LIN {X 0,Y 524.018,Z 138.211,A -85,B 0,C 180,E1 -4848.394,E2 -4848.394} C_VEL
LIN {X 0,Y 523.958,Z 138.22,A -85,B 0,C 180,E1 -4851.515,E2 -4851.515} C_VEL
LIN {X 0,Y 524.039,Z 138.205,A -85,B 0,C 180,E1 -4854.613,E2 -4854.613} C_VEL
LIN {X 0,Y 524.109,Z 138.203,A -85,B 0,C 180,E1 -4857.695,E2 -4857.695} C_VEL
LIN {X 0,Y 524.104,Z 138.202,A -85,B 0,C 180,E1 -4860,E2 -4860} C_VEL
LIN {X 0,Y 524.038,Z 138.21,A -85,B 0,C 180,E1 -4863.075,E2 -4863.075} C_VEL
LIN {X 0,Y 524.015,Z 138.212,A -85,B 0,C 180,E1 -4866.16,E2 -4866.16} C_VEL
LIN {X 0,Y 524.035,Z 138.323,A -85,B 0,C 180,E1 -4867.829,E2 -4867.829} C_VEL
LIN {X 0,Y 524.468,Z 143.022,A -85,B 0,C 180,E1 -4868.671,E2 -4868.671} C_VEL
LIN {X 0,Y 524.363,Z 158.584,A -85,B 0,C 180,E1 -4871.402,E2 -4871.402} C_VEL
LIN {X 0,Y 524.251,Z 167.062,A -85,B 0,C 180,E1 -4872.903,E2 -4872.903} C_VEL
LIN {X 0,Y 525.963,Z 177.173,A -85,B 0,C 180,E1 -4873.105,E2 -4873.105} C_VEL
LIN {X 0,Y 525.467,Z 274.512,A -85,B 0,C 180,E1 -4874.499,E2 -4874.499} C_VEL
LIN {X 0,Y 525.258,Z 287.533,A -85,B 0,C 180,E1 -4874.837,E2 -4874.837} C_VEL
LIN {X 0,Y 525.076,Z 300.224,A -85,B 0,C 180,E1 -4875.326,E2 -4875.326} C_VEL
LIN {X 0,Y 524.793,Z 311.875,A -85,B 0,C 180,E1 -4875.935,E2 -4875.935} C_VEL
LIN {X 0,Y 524.491,Z 323.834,A -85,B 0,C 180,E1 -4876.744,E2 -4876.744} C_VEL
LIN {X 0,Y 524.237,Z 334.197,A -85,B 0,C 180,E1 -4877.625,E2 -4877.625} C_VEL
LIN {X 0,Y 524.02,Z 343.233,A -85,B 0,C 180,E1 -4878.574,E2 -4878.574} C_VEL
LIN {X 0,Y 523.804,Z 351.242,A -85,B 0,C 180,E1 -4879.599,E2 -4879.599} C_VEL
LIN {X 0,Y 523.63,Z 359.058,A -85,B 0,C 180,E1 -4880.835,E2 -4880.835} C_VEL
LIN {X 0,Y 523.487,Z 365.471,A -85,B 0,C 180,E1 -4882.126,E2 -4882.126} C_VEL
LIN {X 0,Y 523.444,Z 370.082,A -85,B 0,C 180,E1 -4883.334,E2 -4883.334} C_VEL
LIN {X 0,Y 523.363,Z 373.668,A -85,B 0,C 180,E1 -4884.601,E2 -4884.601} C_VEL
LIN {X 0,Y 523.278,Z 376.084,A -85,B 0,C 180,E1 -4885.86,E2 -4885.86} C_VEL
LIN {X 0,Y 523.276,Z 377.541,A -85,B 0,C 180,E1 -4887.42,E2 -4887.42} C_VEL
LIN {X 0,Y 522.601,Z 377.718,A -85,B 0,C 180,E1 -4888.062,E2 -4888.062} C_VEL
LIN {X 0,Y 519.728,Z 377.402,A -85,B 0,C 180,E1 -4889.105,E2 -4889.105} C_VEL
LIN {X 0,Y 517.322,Z 376.67,A -85,B 0,C 180,E1 -4889.941,E2 -4889.941} C_VEL
LIN {X 0,Y 516.264,Z 375.561,A -85,B 0,C 180,E1 -4890.691,E2 -4890.691} C_VEL
LIN {X 0,Y 516.251,Z 375.333,A -85,B 0,C 180,E1 -4890.799,E2 -4890.799} C_VEL
LIN {X 0,Y 516.301,Z 372.483,A -85,B 0,C 180,E1 -4892.065,E2 -4892.065} C_VEL
LIN {X 0,Y 516.353,Z 368.046,A -85,B 0,C 180,E1 -4893.436,E2 -4893.436} C_VEL
LIN {X 0,Y 516.459,Z 362.961,A -85,B 0,C 180,E1 -4894.621,E2 -4894.621} C_VEL
LIN {X 0,Y 516.626,Z 356.582,A -85,B 0,C 180,E1 -4895.8,E2 -4895.8} C_VEL
LIN {X 0,Y 516.846,Z 348.507,A -85,B 0,C 180,E1 -4896.993,E2 -4896.993} C_VEL
LIN {X 0,Y 517.108,Z 339.432,A -85,B 0,C 180,E1 -4898.077,E2 -4898.077} C_VEL
LIN {X 0,Y 517.351,Z 330.008,A -85,B 0,C 180,E1 -4898.996,E2 -4898.996} C_VEL
LIN {X 0,Y 517.575,Z 320.063,A -85,B 0,C 180,E1 -4899.785,E2 -4899.785} C_VEL
LIN {X 0,Y 517.926,Z 307.968,A -85,B 0,C 180,E1 -4900.545,E2 -4900.545} C_VEL
LIN {X 0,Y 518.248,Z 295.886,A -85,B 0,C 180,E1 -4901.126,E2 -4901.126} C_VEL
LIN {X 0,Y 518.426,Z 282.731,A -85,B 0,C 180,E1 -4901.578,E2 -4901.578} C_VEL
LIN {X 0,Y 518.601,Z 269.587,A -85,B 0,C 180,E1 -4901.862,E2 -4901.862} C_VEL
LIN {X 0,Y 519.056,Z 177.123,A -85,B 0,C 180,E1 -4903.192,E2 -4903.192} C_VEL
LIN {X 0,Y 517.245,Z 167.202,A -85,B 0,C 180,E1 -4903.401,E2 -4903.401} C_VEL
LIN {X 0,Y 517.6,Z 151.206,A -85,B 0,C 180,E1 -4906.433,E2 -4906.433} C_VEL
LIN {X 0,Y 517.694,Z 144.207,A -85,B 0,C 180,E1 -4907.778,E2 -4907.778} C_VEL
LIN {X 0,Y 516.916,Z 139.099,A -85,B 0,C 180,E1 -4908.846,E2 -4908.846} C_VEL
LIN {X 0,Y 516.881,Z 139.099,A -85,B 0,C 180,E1 -4912.058,E2 -4912.058} C_VEL
LIN {X 0,Y 516.877,Z 139.097,A -85,B 0,C 180,E1 -4915.174,E2 -4915.174} C_VEL
LIN {X 0,Y 516.872,Z 139.098,A -85,B 0,C 180,E1 -4917.974,E2 -4917.974} C_VEL
LIN {X 0,Y 516.84,Z 139.105,A -85,B 0,C 180,E1 -4920.69,E2 -4920.69} C_VEL
LIN {X 0,Y 516.839,Z 139.1,A -85,B 0,C 180,E1 -4923.337,E2 -4923.337} C_VEL
LIN {X 0,Y 516.872,Z 139.1,A -85,B 0,C 180,E1 -4925.925,E2 -4925.925} C_VEL
LIN {X 0,Y 516.858,Z 139.104,A -85,B 0,C 180,E1 -4928.46,E2 -4928.46} C_VEL
LIN {X 0,Y 516.868,Z 139.097,A -85,B 0,C 180,E1 -4930.953,E2 -4930.953} C_VEL
LIN {X 0,Y 516.835,Z 139.101,A -85,B 0,C 180,E1 -4933.407,E2 -4933.407} C_VEL
LIN {X 0,Y 516.876,Z 139.101,A -85,B 0,C 180,E1 -4935.832,E2 -4935.832} C_VEL
LIN {X 0,Y 516.931,Z 139.095,A -85,B 0,C 180,E1 -4938.232,E2 -4938.232} C_VEL
LIN {X 0,Y 516.925,Z 139.091,A -85,B 0,C 180,E1 -4941.398,E2 -4941.398} C_VEL
LIN {X 0,Y 516.984,Z 139.083,A -85,B 0,C 180,E1 -4944.539,E2 -4944.539} C_VEL
LIN {X 0,Y 517.077,Z 139.077,A -85,B 0,C 180,E1 -4947.662,E2 -4947.662} C_VEL
LIN {X 0,Y 517.069,Z 139.078,A -85,B 0,C 180,E1 -4949.999,E2 -4949.999} C_VEL
LIN {X 0,Y 517.076,Z 139.072,A -85,B 0,C 180,E1 -4952.336,E2 -4952.336} C_VEL
LIN {X 0,Y 516.982,Z 139.088,A -85,B 0,C 180,E1 -4955.46,E2 -4955.46} C_VEL
LIN {X 0,Y 516.923,Z 139.09,A -85,B 0,C 180,E1 -4958.6,E2 -4958.6} C_VEL
LIN {X 0,Y 516.936,Z 139.094,A -85,B 0,C 180,E1 -4961.795,E2 -4961.795} C_VEL
LIN {X 0,Y 516.938,Z 139.092,A -85,B 0,C 180,E1 -4965.141,E2 -4965.141} C_VEL
LIN {X 0,Y 516.872,Z 139.096,A -85,B 0,C 180,E1 -4968.223,E2 -4968.223} C_VEL
LIN {X 0,Y 516.872,Z 139.097,A -85,B 0,C 180,E1 -4970.702,E2 -4970.702} C_VEL
LIN {X 0,Y 516.841,Z 139.108,A -85,B 0,C 180,E1 -4973.224,E2 -4973.224} C_VEL
LIN {X 0,Y 516.879,Z 139.095,A -85,B 0,C 180,E1 -4976.18,E2 -4976.18} C_VEL
LIN {X 0,Y 516.896,Z 139.101,A -85,B 0,C 180,E1 -4979.305,E2 -4979.305} C_VEL
LIN {X 0,Y 516.891,Z 139.095,A -85,B 0,C 180,E1 -4982.541,E2 -4982.541} C_VEL
LIN {X 0,Y 516.852,Z 139.104,A -85,B 0,C 180,E1 -4985.327,E2 -4985.327} C_VEL
LIN {X 0,Y 516.875,Z 139.096,A -85,B 0,C 180,E1 -4987.941,E2 -4987.941} C_VEL
LIN {X 0,Y 516.847,Z 139.105,A -85,B 0,C 180,E1 -4990.744,E2 -4990.744} C_VEL
LIN {X 0,Y 516.877,Z 139.095,A -85,B 0,C 180,E1 -4993.903,E2 -4993.903} C_VEL
LIN {X 0,Y 516.876,Z 139.096,A -85,B 0,C 180,E1 -4996.106,E2 -4996.106} C_VEL
LIN {X 0,Y 516.843,Z 139.102,A -85,B 0,C 180,E1 -4999.254,E2 -4999.254} C_VEL
LIN {X 0,Y 516.871,Z 139.097,A -85,B 0,C 180,E1 -5002.057,E2 -5002.057} C_VEL
LIN {X 0,Y 516.866,Z 139.099,A -85,B 0,C 180,E1 -5005.173,E2 -5005.173} C_VEL
LIN {X 0,Y 516.861,Z 139.099,A -85,B 0,C 180,E1 -5007.974,E2 -5007.974} C_VEL
LIN {X 0,Y 516.891,Z 139.1,A -85,B 0,C 180,E1 -5010.693,E2 -5010.693} C_VEL
LIN {X 0,Y 516.873,Z 139.097,A -85,B 0,C 180,E1 -5013.818,E2 -5013.818} C_VEL
LIN {X 0,Y 516.835,Z 139.105,A -85,B 0,C 180,E1 -5016.774,E2 -5016.774} C_VEL
LIN {X 0,Y 516.9,Z 139.094,A -85,B 0,C 180,E1 -5019.741,E2 -5019.741} C_VEL
LIN {X 0,Y 516.861,Z 139.102,A -85,B 0,C 180,E1 -5022.593,E2 -5022.593} C_VEL
LIN {X 0,Y 516.923,Z 139.09,A -85,B 0,C 180,E1 -5025.029,E2 -5025.029} C_VEL
LIN {X 0,Y 516.918,Z 139.099,A -85,B 0,C 180,E1 -5028.232,E2 -5028.232} C_VEL
LIN {X 0,Y 516.912,Z 139.092,A -85,B 0,C 180,E1 -5031.398,E2 -5031.398} C_VEL
LIN {X 0,Y 516.976,Z 139.086,A -85,B 0,C 180,E1 -5034.539,E2 -5034.539} C_VEL
LIN {X 0,Y 517.066,Z 139.076,A -85,B 0,C 180,E1 -5037.663,E2 -5037.663} C_VEL
LIN {X 0,Y 517.057,Z 139.081,A -85,B 0,C 180,E1 -5040,E2 -5040} C_VEL
LIN {X 0,Y 517.065,Z 139.075,A -85,B 0,C 180,E1 -5042.337,E2 -5042.337} C_VEL
LIN {X 0,Y 516.96,Z 139.088,A -85,B 0,C 180,E1 -5046.244,E2 -5046.244} C_VEL
LIN {X 0,Y 516.898,Z 139.097,A -85,B 0,C 180,E1 -5049.39,E2 -5049.39} C_VEL
LIN {X 0,Y 516.888,Z 139.094,A -85,B 0,C 180,E1 -5052.565,E2 -5052.565} C_VEL
LIN {X 0,Y 516.927,Z 139.092,A -85,B 0,C 180,E1 -5055.142,E2 -5055.142} C_VEL
LIN {X 0,Y 516.861,Z 139.098,A -85,B 0,C 180,E1 -5058.224,E2 -5058.224} C_VEL
LIN {X 0,Y 516.862,Z 139.098,A -85,B 0,C 180,E1 -5060.704,E2 -5060.704} C_VEL
LIN {X 0,Y 516.831,Z 139.107,A -85,B 0,C 180,E1 -5063.225,E2 -5063.225} C_VEL
LIN {X 0,Y 516.87,Z 139.097,A -85,B 0,C 180,E1 -5066.181,E2 -5066.181} C_VEL
LIN {X 0,Y 516.821,Z 139.102,A -85,B 0,C 180,E1 -5068.421,E2 -5068.421} C_VEL
LIN {X 0,Y 516.84,Z 139.106,A -85,B 0,C 180,E1 -5071.113,E2 -5071.113} C_VEL
LIN {X 0,Y 516.873,Z 139.097,A -85,B 0,C 180,E1 -5073.962,E2 -5073.962} C_VEL
LIN {X 0,Y 516.808,Z 139.107,A -85,B 0,C 180,E1 -5076.752,E2 -5076.752} C_VEL
LIN {X 0,Y 516.849,Z 139.1,A -85,B 0,C 180,E1 -5079.724,E2 -5079.724} C_VEL
LIN {X 0,Y 516.835,Z 139.106,A -85,B 0,C 180,E1 -5082.837,E2 -5082.837} C_VEL
LIN {X 0,Y 516.89,Z 139.103,A -85,B 0,C 180,E1 -5085.008,E2 -5085.008} C_VEL
LIN {X 0,Y 516.842,Z 139.102,A -85,B 0,C 180,E1 -5088.408,E2 -5088.408} C_VEL
LIN {X 0,Y 516.863,Z 139.1,A -85,B 0,C 180,E1 -5091.284,E2 -5091.284} C_VEL
LIN {X 0,Y 516.844,Z 139.107,A -85,B 0,C 180,E1 -5094.674,E2 -5094.674} C_VEL
LIN {X 0,Y 516.863,Z 139.098,A -85,B 0,C 180,E1 -5097.463,E2 -5097.463} C_VEL
LIN {X 0,Y 516.834,Z 139.108,A -85,B 0,C 180,E1 -5100.492,E2 -5100.492} C_VEL
LIN {X 0,Y 516.829,Z 139.105,A -85,B 0,C 180,E1 -5103.338,E2 -5103.338} C_VEL
LIN {X 0,Y 516.887,Z 139.245,A -85,B 0,C 180,E1 -5105.689,E2 -5105.689} C_VEL
LIN {X 0,Y 518.362,Z 147.957,A -85,B 0,C 180,E1 -5107.213,E2 -5107.213} C_VEL
LIN {X 0,Y 517.967,Z 164.813,A -85,B 0,C 180,E1 -5109.975,E2 -5109.975} C_VEL
LIN {X 0,Y 517.491,Z 183.732,A -85,B 0,C 180,E1 -5113.024,E2 -5113.024} C_VEL
LIN {X 0,Y 517.26,Z 194.139,A -85,B 0,C 180,E1 -5114.646,E2 -5114.646} C_VEL
LIN {X 0,Y 518.975,Z 205.188,A -85,B 0,C 180,E1 -5114.86,E2 -5114.86} C_VEL
LIN {X 0,Y 518.55,Z 301.82,A -85,B 0,C 180,E1 -5116.256,E2 -5116.256} C_VEL
LIN {X 0,Y 518.282,Z 315.071,A -85,B 0,C 180,E1 -5116.598,E2 -5116.598} C_VEL
LIN {X 0,Y 518.055,Z 327.249,A -85,B 0,C 180,E1 -5117.066,E2 -5117.066} C_VEL
LIN {X 0,Y 517.752,Z 339.225,A -85,B 0,C 180,E1 -5117.685,E2 -5117.685} C_VEL
LIN {X 0,Y 517.483,Z 350.536,A -85,B 0,C 180,E1 -5118.445,E2 -5118.445} C_VEL
LIN {X 0,Y 517.197,Z 361.119,A -85,B 0,C 180,E1 -5119.331,E2 -5119.331} C_VEL
LIN {X 0,Y 516.924,Z 369.768,A -85,B 0,C 180,E1 -5120.216,E2 -5120.216} C_VEL
LIN {X 0,Y 516.702,Z 377.739,A -85,B 0,C 180,E1 -5121.199,E2 -5121.199} C_VEL
LIN {X 0,Y 516.531,Z 385.528,A -85,B 0,C 180,E1 -5122.377,E2 -5122.377} C_VEL
LIN {X 0,Y 516.384,Z 392.681,A -85,B 0,C 180,E1 -5123.75,E2 -5123.75} C_VEL
LIN {X 0,Y 516.312,Z 397.442,A -85,B 0,C 180,E1 -5124.925,E2 -5124.925} C_VEL
LIN {X 0,Y 516.351,Z 401.081,A -85,B 0,C 180,E1 -5126.098,E2 -5126.098} C_VEL
LIN {X 0,Y 516.282,Z 402.956,A -85,B 0,C 180,E1 -5126.879,E2 -5126.879} C_VEL
LIN {X 0,Y 516.261,Z 404.361,A -85,B 0,C 180,E1 -5127.66,E2 -5127.66} C_VEL
LIN {X 0,Y 516.162,Z 405.969,A -85,B 0,C 180,E1 -5129.221,E2 -5129.221} C_VEL
LIN {X 0,Y 516.159,Z 406.183,A -85,B 0,C 180,E1 -5130.001,E2 -5130.001} C_VEL
LIN {X 0,Y 516.192,Z 405.347,A -85,B 0,C 180,E1 -5131.561,E2 -5131.561} C_VEL
LIN {X 0,Y 516.261,Z 404.34,A -85,B 0,C 180,E1 -5132.341,E2 -5132.341} C_VEL
LIN {X 0,Y 516.282,Z 402.925,A -85,B 0,C 180,E1 -5133.122,E2 -5133.122} C_VEL
LIN {X 0,Y 516.31,Z 399.956,A -85,B 0,C 180,E1 -5134.294,E2 -5134.294} C_VEL
LIN {X 0,Y 516.368,Z 395.937,A -85,B 0,C 180,E1 -5135.468,E2 -5135.468} C_VEL
LIN {X 0,Y 516.463,Z 390.039,A -85,B 0,C 180,E1 -5136.783,E2 -5136.783} C_VEL
LIN {X 0,Y 516.568,Z 382.987,A -85,B 0,C 180,E1 -5138.017,E2 -5138.017} C_VEL
LIN {X 0,Y 516.767,Z 374.592,A -85,B 0,C 180,E1 -5139.196,E2 -5139.196} C_VEL
LIN {X 0,Y 516.988,Z 365.949,A -85,B 0,C 180,E1 -5140.18,E2 -5140.18} C_VEL
LIN {X 0,Y 517.315,Z 355.287,A -85,B 0,C 180,E1 -5141.163,E2 -5141.163} C_VEL
LIN {X 0,Y 517.563,Z 344.395,A -85,B 0,C 180,E1 -5141.974,E2 -5141.974} C_VEL
LIN {X 0,Y 517.885,Z 333.012,A -85,B 0,C 180,E1 -5142.641,E2 -5142.641} C_VEL
LIN {X 0,Y 518.145,Z 320.861,A -85,B 0,C 180,E1 -5143.182,E2 -5143.182} C_VEL
LIN {X 0,Y 518.396,Z 307.676,A -85,B 0,C 180,E1 -5143.6,E2 -5143.6} C_VEL
LIN {X 0,Y 518.58,Z 295.001,A -85,B 0,C 180,E1 -5143.845,E2 -5143.845} C_VEL
LIN {X 0,Y 518.944,Z 204.771,A -85,B 0,C 180,E1 -5145.142,E2 -5145.142} C_VEL
LIN {X 0,Y 517.215,Z 193.411,A -85,B 0,C 180,E1 -5145.369,E2 -5145.369} C_VEL
LIN {X 0,Y 517.695,Z 172.85,A -85,B 0,C 180,E1 -5148.605,E2 -5148.605} C_VEL
LIN {X 0,Y 518.022,Z 154.72,A -85,B 0,C 180,E1 -5151.489,E2 -5151.489} C_VEL
LIN {X 0,Y 518.101,Z 146.04,A -85,B 0,C 180,E1 -5152.893,E2 -5152.893} C_VEL
LIN {X 0,Y 516.868,Z 139.103,A -85,B 0,C 180,E1 -5154.075,E2 -5154.075} C_VEL
LIN {X 0,Y 516.831,Z 139.107,A -85,B 0,C 180,E1 -5156.664,E2 -5156.664} C_VEL
LIN {X 0,Y 516.84,Z 139.107,A -85,B 0,C 180,E1 -5159.509,E2 -5159.509} C_VEL
LIN {X 0,Y 516.87,Z 139.1,A -85,B 0,C 180,E1 -5162.538,E2 -5162.538} C_VEL
LIN {X 0,Y 516.853,Z 139.105,A -85,B 0,C 180,E1 -5165.327,E2 -5165.327} C_VEL
LIN {X 0,Y 516.874,Z 139.102,A -85,B 0,C 180,E1 -5168.717,E2 -5168.717} C_VEL
LIN {X 0,Y 516.848,Z 139.1,A -85,B 0,C 180,E1 -5171.782,E2 -5171.782} C_VEL
LIN {X 0,Y 516.899,Z 139.098,A -85,B 0,C 180,E1 -5175.007,E2 -5175.007} C_VEL
LIN {X 0,Y 516.851,Z 139.102,A -85,B 0,C 180,E1 -5178.407,E2 -5178.407} C_VEL
LIN {X 0,Y 516.876,Z 139.096,A -85,B 0,C 180,E1 -5181.284,E2 -5181.284} C_VEL
LIN {X 0,Y 516.859,Z 139.101,A -85,B 0,C 180,E1 -5184.219,E2 -5184.219} C_VEL
LIN {X 0,Y 516.882,Z 139.098,A -85,B 0,C 180,E1 -5187.052,E2 -5187.052} C_VEL
LIN {X 0,Y 516.849,Z 139.099,A -85,B 0,C 180,E1 -5189.794,E2 -5189.794} C_VEL
LIN {X 0,Y 516.871,Z 139.104,A -85,B 0,C 180,E1 -5192.464,E2 -5192.464} C_VEL
LIN {X 0,Y 516.848,Z 139.1,A -85,B 0,C 180,E1 -5195.069,E2 -5195.069} C_VEL
LIN {X 0,Y 516.873,Z 139.097,A -85,B 0,C 180,E1 -5197.622,E2 -5197.622} C_VEL
LIN {X 0,Y 516.921,Z 139.097,A -85,B 0,C 180,E1 -5200.129,E2 -5200.129} C_VEL
LIN {X 0,Y 516.869,Z 139.1,A -85,B 0,C 180,E1 -5202.594,E2 -5202.594} C_VEL
LIN {X 0,Y 516.944,Z 139.089,A -85,B 0,C 180,E1 -5205.03,E2 -5205.03} C_VEL
LIN {X 0,Y 516.971,Z 139.091,A -85,B 0,C 180,E1 -5208.234,E2 -5208.234} C_VEL
LIN {X 0,Y 516.934,Z 139.093,A -85,B 0,C 180,E1 -5211.399,E2 -5211.399} C_VEL
LIN {X 0,Y 516.99,Z 139.084,A -85,B 0,C 180,E1 -5214.54,E2 -5214.54} C_VEL
LIN {X 0,Y 517.078,Z 139.079,A -85,B 0,C 180,E1 -5217.663,E2 -5217.663} C_VEL
LIN {X 0,Y 517.072,Z 139.078,A -85,B 0,C 180,E1 -5220,E2 -5220} C_VEL
LIN {X 0,Y 517.083,Z 139.074,A -85,B 0,C 180,E1 -5222.337,E2 -5222.337} C_VEL
LIN {X 0,Y 517.015,Z 139.087,A -85,B 0,C 180,E1 -5225.46,E2 -5225.46} C_VEL
LIN {X 0,Y 517.014,Z 139.25,A -85,B 0,C 180,E1 -5227.715,E2 -5227.715} C_VEL
LIN {X 0,Y 517.492,Z 144.098,A -85,B 0,C 180,E1 -5228.592,E2 -5228.592} C_VEL
LIN {X 0,Y 517.391,Z 158.648,A -85,B 0,C 180,E1 -5231.161,E2 -5231.161} C_VEL
LIN {X 0,Y 517.259,Z 167.216,A -85,B 0,C 180,E1 -5232.688,E2 -5232.688} C_VEL
LIN {X 0,Y 519.12,Z 178.22,A -85,B 0,C 180,E1 -5232.919,E2 -5232.919} C_VEL
LIN {X 0,Y 518.548,Z 274.512,A -85,B 0,C 180,E1 -5234.321,E2 -5234.321} C_VEL
LIN {X 0,Y 518.372,Z 287.213,A -85,B 0,C 180,E1 -5234.652,E2 -5234.652} C_VEL
LIN {X 0,Y 518.159,Z 298.618,A -85,B 0,C 180,E1 -5235.084,E2 -5235.084} C_VEL
LIN {X 0,Y 517.918,Z 309.93,A -85,B 0,C 180,E1 -5235.655,E2 -5235.655} C_VEL
LIN {X 0,Y 517.638,Z 320.905,A -85,B 0,C 180,E1 -5236.363,E2 -5236.363} C_VEL
LIN {X 0,Y 517.317,Z 331.088,A -85,B 0,C 180,E1 -5237.187,E2 -5237.187} C_VEL
LIN {X 0,Y 517.068,Z 341.353,A -85,B 0,C 180,E1 -5238.217,E2 -5238.217} C_VEL
LIN {X 0,Y 516.837,Z 349.758,A -85,B 0,C 180,E1 -5239.254,E2 -5239.254} C_VEL
LIN {X 0,Y 516.625,Z 357.334,A -85,B 0,C 180,E1 -5240.406,E2 -5240.406} C_VEL
LIN {X 0,Y 516.465,Z 363.425,A -85,B 0,C 180,E1 -5241.556,E2 -5241.556} C_VEL
LIN {X 0,Y 516.363,Z 368.714,A -85,B 0,C 180,E1 -5242.824,E2 -5242.824} C_VEL
LIN {X 0,Y 516.281,Z 373.025,A -85,B 0,C 180,E1 -5244.208,E2 -5244.208} C_VEL
LIN {X 0,Y 516.236,Z 374.785,A -85,B 0,C 180,E1 -5244.963,E2 -5244.963} C_VEL
LIN {X 0,Y 516.172,Z 376.548,A -85,B 0,C 180,E1 -5246.02,E2 -5246.02} C_VEL
LIN {X 0,Y 516.179,Z 377.719,A -85,B 0,C 180,E1 -5247.422,E2 -5247.422} C_VEL
LIN {X 0,Y 516.187,Z 377.813,A -85,B 0,C 180,E1 -5248.46,E2 -5248.46} C_VEL
LIN {X 0,Y 516.247,Z 377.281,A -85,B 0,C 180,E1 -5249.392,E2 -5249.392} C_VEL
LIN {X 0,Y 516.251,Z 375.333,A -85,B 0,C 180,E1 -5250.799,E2 -5250.799} C_VEL
LIN {X 0,Y 515.62,Z 374.115,A -85,B 0,C 180,E1 -5251.437,E2 -5251.437} C_VEL
LIN {X 0,Y 512.778,Z 371.571,A -85,B 0,C 180,E1 -5252.457,E2 -5252.457} C_VEL
LIN {X 0,Y 510.391,Z 369.044,A -85,B 0,C 180,E1 -5253.261,E2 -5253.261} C_VEL
LIN {X 0,Y 509.413,Z 366.807,A -85,B 0,C 180,E1 -5253.869,E2 -5253.869} C_VEL
LIN {X 0,Y 509.362,Z 365.974,A -85,B 0,C 180,E1 -5254.072,E2 -5254.072} C_VEL
LIN {X 0,Y 509.528,Z 359.589,A -85,B 0,C 180,E1 -5255.403,E2 -5255.403} C_VEL
LIN {X 0,Y 509.71,Z 352.041,A -85,B 0,C 180,E1 -5256.638,E2 -5256.638} C_VEL
LIN {X 0,Y 509.977,Z 343.015,A -85,B 0,C 180,E1 -5257.826,E2 -5257.826} C_VEL
LIN {X 0,Y 510.243,Z 333.745,A -85,B 0,C 180,E1 -5258.808,E2 -5258.808} C_VEL
LIN {X 0,Y 510.548,Z 323.768,A -85,B 0,C 180,E1 -5259.67,E2 -5259.67} C_VEL
LIN {X 0,Y 510.839,Z 313.416,A -85,B 0,C 180,E1 -5260.395,E2 -5260.395} C_VEL
LIN {X 0,Y 511.184,Z 301.901,A -85,B 0,C 180,E1 -5261.033,E2 -5261.033} C_VEL
LIN {X 0,Y 511.397,Z 289.381,A -85,B 0,C 180,E1 -5261.553,E2 -5261.553} C_VEL
LIN {X 0,Y 511.625,Z 276.213,A -85,B 0,C 180,E1 -5261.921,E2 -5261.921} C_VEL
LIN {X 0,Y 511.782,Z 249.363,A -85,B 0,C 180,E1 -5262.341,E2 -5262.341} C_VEL
LIN {X 0,Y 512.117,Z 177.423,A -85,B 0,C 180,E1 -5263.396,E2 -5263.396} C_VEL
LIN {X 0,Y 510.268,Z 167.314,A -85,B 0,C 180,E1 -5263.623,E2 -5263.623} C_VEL
LIN {X 0,Y 510.689,Z 150.589,A -85,B 0,C 180,E1 -5266.835,E2 -5266.835} C_VEL
LIN {X 0,Y 510.672,Z 144.608,A -85,B 0,C 180,E1 -5268.002,E2 -5268.002} C_VEL
LIN {X 0,Y 509.874,Z 139.976,A -85,B 0,C 180,E1 -5268.976,E2 -5268.976} C_VEL
LIN {X 0,Y 509.827,Z 139.976,A -85,B 0,C 180,E1 -5271.791,E2 -5271.791} C_VEL
LIN {X 0,Y 509.824,Z 139.982,A -85,B 0,C 180,E1 -5274.621,E2 -5274.621} C_VEL
LIN {X 0,Y 509.863,Z 139.969,A -85,B 0,C 180,E1 -5277.48,E2 -5277.48} C_VEL
LIN {X 0,Y 509.796,Z 139.984,A -85,B 0,C 180,E1 -5280.287,E2 -5280.287} C_VEL
LIN {X 0,Y 509.824,Z 139.976,A -85,B 0,C 180,E1 -5282.94,E2 -5282.94} C_VEL
LIN {X 0,Y 509.827,Z 139.974,A -85,B 0,C 180,E1 -5285.571,E2 -5285.571} C_VEL
LIN {X 0,Y 509.808,Z 139.983,A -85,B 0,C 180,E1 -5288.147,E2 -5288.147} C_VEL
LIN {X 0,Y 509.83,Z 139.976,A -85,B 0,C 180,E1 -5290.68,E2 -5290.68} C_VEL
LIN {X 0,Y 509.79,Z 139.978,A -85,B 0,C 180,E1 -5293.171,E2 -5293.171} C_VEL
LIN {X 0,Y 509.849,Z 139.973,A -85,B 0,C 180,E1 -5295.633,E2 -5295.633} C_VEL
LIN {X 0,Y 509.895,Z 139.973,A -85,B 0,C 180,E1 -5298.13,E2 -5298.13} C_VEL
LIN {X 0,Y 509.878,Z 139.968,A -85,B 0,C 180,E1 -5301.278,E2 -5301.278} C_VEL
LIN {X 0,Y 509.92,Z 139.967,A -85,B 0,C 180,E1 -5303.669,E2 -5303.669} C_VEL
LIN {X 0,Y 509.888,Z 139.966,A -85,B 0,C 180,E1 -5306.839,E2 -5306.839} C_VEL
LIN {X 0,Y 509.926,Z 139.963,A -85,B 0,C 180,E1 -5308.42,E2 -5308.42} C_VEL
LIN {X 0,Y 510.038,Z 139.953,A -85,B 0,C 180,E1 -5309.999,E2 -5309.999} C_VEL
LIN {X 0,Y 510.044,Z 139.948,A -85,B 0,C 180,E1 -5312.368,E2 -5312.368} C_VEL
LIN {X 0,Y 509.935,Z 139.967,A -85,B 0,C 180,E1 -5315.536,E2 -5315.536} C_VEL
LIN {X 0,Y 509.878,Z 139.972,A -85,B 0,C 180,E1 -5317.922,E2 -5317.922} C_VEL
LIN {X 0,Y 509.864,Z 139.972,A -85,B 0,C 180,E1 -5321.126,E2 -5321.126} C_VEL
LIN {X 0,Y 509.842,Z 139.972,A -85,B 0,C 180,E1 -5324.366,E2 -5324.366} C_VEL
LIN {X 0,Y 509.798,Z 139.979,A -85,B 0,C 180,E1 -5326.827,E2 -5326.827} C_VEL
LIN {X 0,Y 509.827,Z 139.981,A -85,B 0,C 180,E1 -5329.319,E2 -5329.319} C_VEL
LIN {X 0,Y 509.825,Z 139.974,A -85,B 0,C 180,E1 -5332.54,E2 -5332.54} C_VEL
LIN {X 0,Y 509.8,Z 139.986,A -85,B 0,C 180,E1 -5335.299,E2 -5335.299} C_VEL
LIN {X 0,Y 509.81,Z 139.976,A -85,B 0,C 180,E1 -5338.081,E2 -5338.081} C_VEL
LIN {X 0,Y 509.803,Z 139.979,A -85,B 0,C 180,E1 -5340.668,E2 -5340.668} C_VEL
LIN {X 0,Y 509.837,Z 139.976,A -85,B 0,C 180,E1 -5343.462,E2 -5343.462} C_VEL
LIN {X 0,Y 509.801,Z 139.978,A -85,B 0,C 180,E1 -5346.354,E2 -5346.354} C_VEL
LIN {X 0,Y 509.829,Z 139.977,A -85,B 0,C 180,E1 -5349.353,E2 -5349.353} C_VEL
LIN {X 0,Y 509.786,Z 139.982,A -85,B 0,C 180,E1 -5352.494,E2 -5352.494} C_VEL
LIN {X 0,Y 509.836,Z 139.975,A -85,B 0,C 180,E1 -5355.329,E2 -5355.329} C_VEL
LIN {X 0,Y 509.798,Z 139.983,A -85,B 0,C 180,E1 -5358.568,E2 -5358.568} C_VEL
LIN {X 0,Y 509.816,Z 139.975,A -85,B 0,C 180,E1 -5361.658,E2 -5361.658} C_VEL
LIN {X 0,Y 509.813,Z 139.984,A -85,B 0,C 180,E1 -5364.62,E2 -5364.62} C_VEL
LIN {X 0,Y 509.852,Z 139.971,A -85,B 0,C 180,E1 -5367.48,E2 -5367.48} C_VEL
LIN {X 0,Y 509.821,Z 139.979,A -85,B 0,C 180,E1 -5370.279,E2 -5370.279} C_VEL
LIN {X 0,Y 509.812,Z 139.978,A -85,B 0,C 180,E1 -5372.94,E2 -5372.94} C_VEL
LIN {X 0,Y 509.827,Z 139.974,A -85,B 0,C 180,E1 -5375.571,E2 -5375.571} C_VEL
LIN {X 0,Y 509.803,Z 139.982,A -85,B 0,C 180,E1 -5378.147,E2 -5378.147} C_VEL
LIN {X 0,Y 509.837,Z 139.977,A -85,B 0,C 180,E1 -5380.68,E2 -5380.68} C_VEL
LIN {X 0,Y 509.782,Z 139.979,A -85,B 0,C 180,E1 -5383.171,E2 -5383.171} C_VEL
LIN {X 0,Y 509.836,Z 139.974,A -85,B 0,C 180,E1 -5385.633,E2 -5385.633} C_VEL
LIN {X 0,Y 509.882,Z 139.975,A -85,B 0,C 180,E1 -5388.13,E2 -5388.13} C_VEL
LIN {X 0,Y 509.865,Z 139.969,A -85,B 0,C 180,E1 -5391.279,E2 -5391.279} C_VEL
LIN {X 0,Y 509.914,Z 139.966,A -85,B 0,C 180,E1 -5393.669,E2 -5393.669} C_VEL
LIN {X 0,Y 509.877,Z 139.968,A -85,B 0,C 180,E1 -5396.839,E2 -5396.839} C_VEL
LIN {X 0,Y 509.914,Z 139.966,A -85,B 0,C 180,E1 -5398.42,E2 -5398.42} C_VEL
LIN {X 0,Y 510.026,Z 139.957,A -85,B 0,C 180,E1 -5400,E2 -5400} C_VEL
LIN {X 0,Y 510.033,Z 139.95,A -85,B 0,C 180,E1 -5402.369,E2 -5402.369} C_VEL
LIN {X 0,Y 509.927,Z 139.966,A -85,B 0,C 180,E1 -5405.536,E2 -5405.536} C_VEL
LIN {X 0,Y 509.866,Z 139.976,A -85,B 0,C 180,E1 -5407.923,E2 -5407.923} C_VEL
LIN {X 0,Y 509.853,Z 139.972,A -85,B 0,C 180,E1 -5411.127,E2 -5411.127} C_VEL
LIN {X 0,Y 509.815,Z 139.983,A -85,B 0,C 180,E1 -5413.553,E2 -5413.553} C_VEL
LIN {X 0,Y 509.795,Z 139.981,A -85,B 0,C 180,E1 -5416.005,E2 -5416.005} C_VEL
LIN {X 0,Y 509.818,Z 139.975,A -85,B 0,C 180,E1 -5418.485,E2 -5418.485} C_VEL
LIN {X 0,Y 509.809,Z 139.978,A -85,B 0,C 180,E1 -5421.003,E2 -5421.003} C_VEL
LIN {X 0,Y 509.794,Z 139.985,A -85,B 0,C 180,E1 -5423.565,E2 -5423.565} C_VEL
LIN {X 0,Y 509.806,Z 139.976,A -85,B 0,C 180,E1 -5426.356,E2 -5426.356} C_VEL
LIN {X 0,Y 509.785,Z 139.981,A -85,B 0,C 180,E1 -5428.85,E2 -5428.85} C_VEL
LIN {X 0,Y 509.789,Z 139.983,A -85,B 0,C 180,E1 -5431.592,E2 -5431.592} C_VEL
LIN {X 0,Y 509.825,Z 139.974,A -85,B 0,C 180,E1 -5434.415,E2 -5434.415} C_VEL
LIN {X 0,Y 509.775,Z 139.986,A -85,B 0,C 180,E1 -5437.344,E2 -5437.344} C_VEL
LIN {X 0,Y 509.805,Z 139.977,A -85,B 0,C 180,E1 -5440.385,E2 -5440.385} C_VEL
LIN {X 0,Y 509.786,Z 139.981,A -85,B 0,C 180,E1 -5443.575,E2 -5443.575} C_VEL
LIN {X 0,Y 509.786,Z 139.981,A -85,B 0,C 180,E1 -5446.426,E2 -5446.426} C_VEL
LIN {X 0,Y 509.806,Z 139.977,A -85,B 0,C 180,E1 -5449.616,E2 -5449.616} C_VEL
LIN {X 0,Y 509.774,Z 139.986,A -85,B 0,C 180,E1 -5452.657,E2 -5452.657} C_VEL
LIN {X 0,Y 509.834,Z 139.973,A -85,B 0,C 180,E1 -5455.801,E2 -5455.801} C_VEL
LIN {X 0,Y 509.811,Z 139.985,A -85,B 0,C 180,E1 -5458.727,E2 -5458.727} C_VEL
LIN {X 0,Y 509.819,Z 139.977,A -85,B 0,C 180,E1 -5462.051,E2 -5462.051} C_VEL
LIN {X 0,Y 509.792,Z 139.987,A -85,B 0,C 180,E1 -5464.7,E2 -5464.7} C_VEL
LIN {X 0,Y 509.844,Z 140.159,A -85,B 0,C 180,E1 -5465.517,E2 -5465.517} C_VEL
LIN {X 0,Y 511.398,Z 148.702,A -85,B 0,C 180,E1 -5467.038,E2 -5467.038} C_VEL
LIN {X 0,Y 511.037,Z 164.827,A -85,B 0,C 180,E1 -5469.722,E2 -5469.722} C_VEL
LIN {X 0,Y 510.53,Z 181.024,A -85,B 0,C 180,E1 -5472.372,E2 -5472.372} C_VEL
LIN {X 0,Y 510.229,Z 193.684,A -85,B 0,C 180,E1 -5474.423,E2 -5474.423} C_VEL
LIN {X 0,Y 512.14,Z 206.103,A -85,B 0,C 180,E1 -5474.669,E2 -5474.669} C_VEL
LIN {X 0,Y 511.608,Z 302.384,A -85,B 0,C 180,E1 -5476.091,E2 -5476.091} C_VEL
LIN {X 0,Y 511.336,Z 316.131,A -85,B 0,C 180,E1 -5476.463,E2 -5476.463} C_VEL
LIN {X 0,Y 511.1,Z 327.987,A -85,B 0,C 180,E1 -5476.937,E2 -5476.937} C_VEL
LIN {X 0,Y 510.717,Z 340.754,A -85,B 0,C 180,E1 -5477.631,E2 -5477.631} C_VEL
LIN {X 0,Y 510.44,Z 352.83,A -85,B 0,C 180,E1 -5478.485,E2 -5478.485} C_VEL
LIN {X 0,Y 510.156,Z 361.913,A -85,B 0,C 180,E1 -5479.283,E2 -5479.283} C_VEL
LIN {X 0,Y 509.829,Z 371.228,A -85,B 0,C 180,E1 -5480.279,E2 -5480.279} C_VEL
LIN {X 0,Y 509.605,Z 380.27,A -85,B 0,C 180,E1 -5481.475,E2 -5481.475} C_VEL
LIN {X 0,Y 509.426,Z 387.551,A -85,B 0,C 180,E1 -5482.669,E2 -5482.669} C_VEL
LIN {X 0,Y 509.307,Z 392.463,A -85,B 0,C 180,E1 -5483.663,E2 -5483.663} C_VEL
LIN {X 0,Y 509.241,Z 397.233,A -85,B 0,C 180,E1 -5484.854,E2 -5484.854} C_VEL
LIN {X 0,Y 509.244,Z 400.878,A -85,B 0,C 180,E1 -5486.044,E2 -5486.044} C_VEL
LIN {X 0,Y 509.2,Z 402.757,A -85,B 0,C 180,E1 -5486.836,E2 -5486.836} C_VEL
LIN {X 0,Y 509.19,Z 404.166,A -85,B 0,C 180,E1 -5487.628,E2 -5487.628} C_VEL
LIN {X 0,Y 509.076,Z 405.775,A -85,B 0,C 180,E1 -5489.21,E2 -5489.21} C_VEL
LIN {X 0,Y 509.07,Z 405.989,A -85,B 0,C 180,E1 -5490.001,E2 -5490.001} C_VEL
LIN {X 0,Y 509.076,Z 405.766,A -85,B 0,C 180,E1 -5490.792,E2 -5490.792} C_VEL
LIN {X 0,Y 509.19,Z 404.138,A -85,B 0,C 180,E1 -5492.374,E2 -5492.374} C_VEL
LIN {X 0,Y 509.2,Z 402.719,A -85,B 0,C 180,E1 -5493.165,E2 -5493.165} C_VEL
LIN {X 0,Y 509.202,Z 399.741,A -85,B 0,C 180,E1 -5494.354,E2 -5494.354} C_VEL
LIN {X 0,Y 509.284,Z 395.712,A -85,B 0,C 180,E1 -5495.544,E2 -5495.544} C_VEL
LIN {X 0,Y 509.403,Z 389.61,A -85,B 0,C 180,E1 -5496.914,E2 -5496.914} C_VEL
LIN {X 0,Y 509.495,Z 382.727,A -85,B 0,C 180,E1 -5498.129,E2 -5498.129} C_VEL
LIN {X 0,Y 509.725,Z 374.313,A -85,B 0,C 180,E1 -5499.324,E2 -5499.324} C_VEL
LIN {X 0,Y 509.959,Z 365.643,A -85,B 0,C 180,E1 -5500.321,E2 -5500.321} C_VEL
LIN {X 0,Y 510.333,Z 354.953,A -85,B 0,C 180,E1 -5501.318,E2 -5501.318} C_VEL
LIN {X 0,Y 510.602,Z 344.045,A -85,B 0,C 180,E1 -5502.138,E2 -5502.138} C_VEL
LIN {X 0,Y 510.966,Z 331.589,A -85,B 0,C 180,E1 -5502.865,E2 -5502.865} C_VEL
LIN {X 0,Y 511.232,Z 319.076,A -85,B 0,C 180,E1 -5503.415,E2 -5503.415} C_VEL
LIN {X 0,Y 511.505,Z 306.101,A -85,B 0,C 180,E1 -5503.812,E2 -5503.812} C_VEL
LIN {X 0,Y 511.716,Z 290.655,A -85,B 0,C 180,E1 -5504.085,E2 -5504.085} C_VEL
LIN {X 0,Y 511.973,Z 204.978,A -85,B 0,C 180,E1 -5505.346,E2 -5505.346} C_VEL
LIN {X 0,Y 510.214,Z 193.187,A -85,B 0,C 180,E1 -5505.587,E2 -5505.587} C_VEL
LIN {X 0,Y 510.699,Z 173.895,A -85,B 0,C 180,E1 -5508.661,E2 -5508.661} C_VEL
LIN {X 0,Y 511.069,Z 155.803,A -85,B 0,C 180,E1 -5511.584,E2 -5511.584} C_VEL
LIN {X 0,Y 511.183,Z 147.73,A -85,B 0,C 180,E1 -5512.905,E2 -5512.905} C_VEL
LIN {X 0,Y 509.812,Z 139.982,A -85,B 0,C 180,E1 -5514.267,E2 -5514.267} C_VEL
LIN {X 0,Y 509.816,Z 139.985,A -85,B 0,C 180,E1 -5517.06,E2 -5517.06} C_VEL
LIN {X 0,Y 509.786,Z 139.983,A -85,B 0,C 180,E1 -5519.756,E2 -5519.756} C_VEL
LIN {X 0,Y 509.829,Z 139.979,A -85,B 0,C 180,E1 -5522.766,E2 -5522.766} C_VEL
LIN {X 0,Y 509.798,Z 139.981,A -85,B 0,C 180,E1 -5525.574,E2 -5525.574} C_VEL
LIN {X 0,Y 509.817,Z 139.977,A -85,B 0,C 180,E1 -5528.342,E2 -5528.342} C_VEL
LIN {X 0,Y 509.806,Z 139.979,A -85,B 0,C 180,E1 -5531.431,E2 -5531.431} C_VEL
LIN {X 0,Y 509.842,Z 139.978,A -85,B 0,C 180,E1 -5534.67,E2 -5534.67} C_VEL
LIN {X 0,Y 509.791,Z 139.978,A -85,B 0,C 180,E1 -5537.506,E2 -5537.506} C_VEL
LIN {X 0,Y 509.833,Z 139.98,A -85,B 0,C 180,E1 -5540.646,E2 -5540.646} C_VEL
LIN {X 0,Y 509.805,Z 139.976,A -85,B 0,C 180,E1 -5543.645,E2 -5543.645} C_VEL
LIN {X 0,Y 509.841,Z 139.979,A -85,B 0,C 180,E1 -5546.538,E2 -5546.538} C_VEL
LIN {X 0,Y 509.823,Z 139.974,A -85,B 0,C 180,E1 -5549.333,E2 -5549.333} C_VEL
LIN {X 0,Y 509.827,Z 139.977,A -85,B 0,C 180,E1 -5552.051,E2 -5552.051} C_VEL
LIN {X 0,Y 509.804,Z 139.98,A -85,B 0,C 180,E1 -5554.7,E2 -5554.7} C_VEL
LIN {X 0,Y 509.828,Z 139.974,A -85,B 0,C 180,E1 -5557.459,E2 -5557.459} C_VEL
LIN {X 0,Y 509.909,Z 139.967,A -85,B 0,C 180,E1 -5559.844,E2 -5559.844} C_VEL
LIN {X 0,Y 509.85,Z 139.978,A -85,B 0,C 180,E1 -5562.347,E2 -5562.347} C_VEL
LIN {X 0,Y 509.893,Z 139.968,A -85,B 0,C 180,E1 -5564.818,E2 -5564.818} C_VEL
LIN {X 0,Y 509.905,Z 139.972,A -85,B 0,C 180,E1 -5568.124,E2 -5568.124} C_VEL
LIN {X 0,Y 509.888,Z 139.97,A -85,B 0,C 180,E1 -5571.279,E2 -5571.279} C_VEL
LIN {X 0,Y 509.944,Z 139.962,A -85,B 0,C 180,E1 -5574.464,E2 -5574.464} C_VEL
LIN {X 0,Y 510.047,Z 139.955,A -85,B 0,C 180,E1 -5577.631,E2 -5577.631} C_VEL
LIN {X 0,Y 510.041,Z 139.954,A -85,B 0,C 180,E1 -5580,E2 -5580} C_VEL
LIN {X 0,Y 510.052,Z 139.95,A -85,B 0,C 180,E1 -5582.369,E2 -5582.369} C_VEL
LIN {X 0,Y 509.966,Z 139.965,A -85,B 0,C 180,E1 -5585.536,E2 -5585.536} C_VEL
LIN {X 0,Y 509.954,Z 140.148,A -85,B 0,C 180,E1 -5587.573,E2 -5587.573} C_VEL
LIN {X 0,Y 510.531,Z 145.232,A -85,B 0,C 180,E1 -5588.51,E2 -5588.51} C_VEL
LIN {X 0,Y 510.395,Z 159.842,A -85,B 0,C 180,E1 -5591.115,E2 -5591.115} C_VEL
LIN {X 0,Y 510.345,Z 167.687,A -85,B 0,C 180,E1 -5592.486,E2 -5592.486} C_VEL
LIN {X 0,Y 512.286,Z 179.682,A -85,B 0,C 180,E1 -5592.73,E2 -5592.73} C_VEL
LIN {X 0,Y 511.657,Z 274.521,A -85,B 0,C 180,E1 -5594.137,E2 -5594.137} C_VEL
LIN {X 0,Y 511.45,Z 287.306,A -85,B 0,C 180,E1 -5594.473,E2 -5594.473} C_VEL
LIN {X 0,Y 511.208,Z 300.471,A -85,B 0,C 180,E1 -5594.989,E2 -5594.989} C_VEL
LIN {X 0,Y 510.892,Z 312.657,A -85,B 0,C 180,E1 -5595.645,E2 -5595.645} C_VEL
LIN {X 0,Y 510.531,Z 324.791,A -85,B 0,C 180,E1 -5596.495,E2 -5596.495} C_VEL
LIN {X 0,Y 510.203,Z 335.385,A -85,B 0,C 180,E1 -5597.434,E2 -5597.434} C_VEL
LIN {X 0,Y 509.939,Z 344.871,A -85,B 0,C 180,E1 -5598.481,E2 -5598.481} C_VEL
LIN {X 0,Y 509.701,Z 352.684,A -85,B 0,C 180,E1 -5599.535,E2 -5599.535} C_VEL
LIN {X 0,Y 509.491,Z 360.378,A -85,B 0,C 180,E1 -5600.818,E2 -5600.818} C_VEL
LIN {X 0,Y 509.331,Z 366.534,A -85,B 0,C 180,E1 -5602.139,E2 -5602.139} C_VEL
LIN {X 0,Y 509.222,Z 371.673,A -85,B 0,C 180,E1 -5603.594,E2 -5603.594} C_VEL
LIN {X 0,Y 509.174,Z 373.956,A -85,B 0,C 180,E1 -5604.462,E2 -5604.462} C_VEL
LIN {X 0,Y 509.11,Z 375.74,A -85,B 0,C 180,E1 -5605.337,E2 -5605.337} C_VEL
LIN {X 0,Y 509.099,Z 377.028,A -85,B 0,C 180,E1 -5606.216,E2 -5606.216} C_VEL
LIN {X 0,Y 509.078,Z 377.787,A -85,B 0,C 180,E1 -5607.102,E2 -5607.102} C_VEL
LIN {X 0,Y 509.089,Z 378.085,A -85,B 0,C 180,E1 -5607.994,E2 -5607.994} C_VEL
LIN {X 0,Y 509.139,Z 377.298,A -85,B 0,C 180,E1 -5609.583,E2 -5609.583} C_VEL
LIN {X 0,Y 509.199,Z 374.951,A -85,B 0,C 180,E1 -5611.159,E2 -5611.159} C_VEL
LIN {X 0,Y 509.228,Z 371.106,A -85,B 0,C 180,E1 -5612.66,E2 -5612.66} C_VEL
LIN {X 0,Y 509.362,Z 365.974,A -85,B 0,C 180,E1 -5614.072,E2 -5614.072} C_VEL
LIN {X 0,Y 508.791,Z 363.434,A -85,B 0,C 180,E1 -5614.669,E2 -5614.669} C_VEL
LIN {X 0,Y 506.069,Z 358.889,A -85,B 0,C 180,E1 -5615.616,E2 -5615.616} C_VEL
LIN {X 0,Y 503.341,Z 353.679,A -85,B 0,C 180,E1 -5616.526,E2 -5616.526} C_VEL
LIN {X 0,Y 502.768,Z 350.094,A -85,B 0,C 180,E1 -5617.059,E2 -5617.059} C_VEL
LIN {X 0,Y 503.02,Z 341.444,A -85,B 0,C 180,E1 -5618.155,E2 -5618.155} C_VEL
LIN {X 0,Y 503.335,Z 331.431,A -85,B 0,C 180,E1 -5619.185,E2 -5619.185} C_VEL
LIN {X 0,Y 503.639,Z 320.826,A -85,B 0,C 180,E1 -5620.065,E2 -5620.065} C_VEL
LIN {X 0,Y 504.019,Z 309.339,A -85,B 0,C 180,E1 -5620.816,E2 -5620.816} C_VEL
LIN {X 0,Y 504.364,Z 297.39,A -85,B 0,C 180,E1 -5621.42,E2 -5621.42} C_VEL
LIN {X 0,Y 504.575,Z 285.264,A -85,B 0,C 180,E1 -5621.873,E2 -5621.873} C_VEL
LIN {X 0,Y 504.774,Z 272.092,A -85,B 0,C 180,E1 -5622.191,E2 -5622.191} C_VEL
LIN {X 0,Y 505.283,Z 178.343,A -85,B 0,C 180,E1 -5623.591,E2 -5623.591} C_VEL
LIN {X 0,Y 503.28,Z 167.512,A -85,B 0,C 180,E1 -5623.833,E2 -5623.833} C_VEL
LIN {X 0,Y 503.768,Z 150.718,A -85,B 0,C 180,E1 -5627.097,E2 -5627.097} C_VEL
LIN {X 0,Y 503.59,Z 145.114,A -85,B 0,C 180,E1 -5628.21,E2 -5628.21} C_VEL
LIN {X 0,Y 502.836,Z 140.852,A -85,B 0,C 180,E1 -5629.114,E2 -5629.114} C_VEL
LIN {X 0,Y 502.777,Z 140.856,A -85,B 0,C 180,E1 -5632.044,E2 -5632.044} C_VEL
LIN {X 0,Y 502.794,Z 140.852,A -85,B 0,C 180,E1 -5635.033,E2 -5635.033} C_VEL
LIN {X 0,Y 502.784,Z 140.853,A -85,B 0,C 180,E1 -5637.915,E2 -5637.915} C_VEL
LIN {X 0,Y 502.763,Z 140.858,A -85,B 0,C 180,E1 -5640.708,E2 -5640.708} C_VEL
LIN {X 0,Y 502.777,Z 140.852,A -85,B 0,C 180,E1 -5643.46,E2 -5643.46} C_VEL
LIN {X 0,Y 502.758,Z 140.86,A -85,B 0,C 180,E1 -5646.084,E2 -5646.084} C_VEL
LIN {X 0,Y 502.764,Z 140.856,A -85,B 0,C 180,E1 -5648.687,E2 -5648.687} C_VEL
LIN {X 0,Y 502.798,Z 140.854,A -85,B 0,C 180,E1 -5651.897,E2 -5651.897} C_VEL
LIN {X 0,Y 502.83,Z 140.846,A -85,B 0,C 180,E1 -5655.428,E2 -5655.428} C_VEL
LIN {X 0,Y 502.842,Z 140.845,A -85,B 0,C 180,E1 -5658.715,E2 -5658.715} C_VEL
LIN {X 0,Y 502.851,Z 140.852,A -85,B 0,C 180,E1 -5661.965,E2 -5661.965} C_VEL
LIN {X 0,Y 502.896,Z 140.84,A -85,B 0,C 180,E1 -5664.385,E2 -5664.385} C_VEL
LIN {X 0,Y 503.013,Z 140.828,A -85,B 0,C 180,E1 -5667.597,E2 -5667.597} C_VEL
LIN {X 0,Y 503.007,Z 140.829,A -85,B 0,C 180,E1 -5669.999,E2 -5669.999} C_VEL
LIN {X 0,Y 503.012,Z 140.824,A -85,B 0,C 180,E1 -5672.402,E2 -5672.402} C_VEL
LIN {X 0,Y 502.891,Z 140.846,A -85,B 0,C 180,E1 -5675.613,E2 -5675.613} C_VEL
LIN {X 0,Y 502.85,Z 140.846,A -85,B 0,C 180,E1 -5678.033,E2 -5678.033} C_VEL
LIN {X 0,Y 502.84,Z 140.849,A -85,B 0,C 180,E1 -5681.283,E2 -5681.283} C_VEL
LIN {X 0,Y 502.824,Z 140.846,A -85,B 0,C 180,E1 -5684.571,E2 -5684.571} C_VEL
LIN {X 0,Y 502.786,Z 140.853,A -85,B 0,C 180,E1 -5687.909,E2 -5687.909} C_VEL
LIN {X 0,Y 502.804,Z 140.849,A -85,B 0,C 180,E1 -5690.527,E2 -5690.527} C_VEL
LIN {X 0,Y 502.782,Z 140.856,A -85,B 0,C 180,E1 -5693.04,E2 -5693.04} C_VEL
LIN {X 0,Y 502.776,Z 140.855,A -85,B 0,C 180,E1 -5695.678,E2 -5695.678} C_VEL
LIN {X 0,Y 502.769,Z 140.853,A -85,B 0,C 180,E1 -5698.376,E2 -5698.376} C_VEL
LIN {X 0,Y 502.764,Z 140.862,A -85,B 0,C 180,E1 -5701.145,E2 -5701.145} C_VEL
LIN {X 0,Y 502.784,Z 140.851,A -85,B 0,C 180,E1 -5703.994,E2 -5703.994} C_VEL
LIN {X 0,Y 502.761,Z 140.861,A -85,B 0,C 180,E1 -5707.174,E2 -5707.174} C_VEL
LIN {X 0,Y 502.768,Z 140.853,A -85,B 0,C 180,E1 -5710.016,E2 -5710.016} C_VEL
LIN {X 0,Y 502.743,Z 140.86,A -85,B 0,C 180,E1 -5713.233,E2 -5713.233} C_VEL
LIN {X 0,Y 502.775,Z 140.853,A -85,B 0,C 180,E1 -5715.659,E2 -5715.659} C_VEL
LIN {X 0,Y 502.758,Z 140.86,A -85,B 0,C 180,E1 -5719.012,E2 -5719.012} C_VEL
LIN {X 0,Y 502.767,Z 140.854,A -85,B 0,C 180,E1 -5722.043,E2 -5722.043} C_VEL
LIN {X 0,Y 502.783,Z 140.855,A -85,B 0,C 180,E1 -5725.032,E2 -5725.032} C_VEL
LIN {X 0,Y 502.773,Z 140.853,A -85,B 0,C 180,E1 -5727.914,E2 -5727.914} C_VEL
LIN {X 0,Y 502.783,Z 140.858,A -85,B 0,C 180,E1 -5730.709,E2 -5730.709} C_VEL
LIN {X 0,Y 502.767,Z 140.853,A -85,B 0,C 180,E1 -5733.459,E2 -5733.459} C_VEL
LIN {X 0,Y 502.754,Z 140.859,A -85,B 0,C 180,E1 -5736.084,E2 -5736.084} C_VEL
LIN {X 0,Y 502.823,Z 140.846,A -85,B 0,C 180,E1 -5739.463,E2 -5739.463} C_VEL
LIN {X 0,Y 502.777,Z 140.857,A -85,B 0,C 180,E1 -5742.09,E2 -5742.09} C_VEL
LIN {X 0,Y 502.817,Z 140.847,A -85,B 0,C 180,E1 -5745.428,E2 -5745.428} C_VEL
LIN {X 0,Y 502.83,Z 140.847,A -85,B 0,C 180,E1 -5748.715,E2 -5748.715} C_VEL
LIN {X 0,Y 502.838,Z 140.851,A -85,B 0,C 180,E1 -5751.965,E2 -5751.965} C_VEL
LIN {X 0,Y 502.888,Z 140.842,A -85,B 0,C 180,E1 -5754.386,E2 -5754.386} C_VEL
LIN {X 0,Y 503.001,Z 140.827,A -85,B 0,C 180,E1 -5757.597,E2 -5757.597} C_VEL
LIN {X 0,Y 502.995,Z 140.833,A -85,B 0,C 180,E1 -5760,E2 -5760} C_VEL
LIN {X 0,Y 503.001,Z 140.826,A -85,B 0,C 180,E1 -5762.402,E2 -5762.402} C_VEL
LIN {X 0,Y 502.884,Z 140.844,A -85,B 0,C 180,E1 -5765.614,E2 -5765.614} C_VEL
LIN {X 0,Y 502.838,Z 140.849,A -85,B 0,C 180,E1 -5768.034,E2 -5768.034} C_VEL
LIN {X 0,Y 502.828,Z 140.849,A -85,B 0,C 180,E1 -5771.284,E2 -5771.284} C_VEL
LIN {X 0,Y 502.815,Z 140.847,A -85,B 0,C 180,E1 -5774.572,E2 -5774.572} C_VEL
LIN {X 0,Y 502.776,Z 140.856,A -85,B 0,C 180,E1 -5777.91,E2 -5777.91} C_VEL
LIN {X 0,Y 502.794,Z 140.85,A -85,B 0,C 180,E1 -5780.528,E2 -5780.528} C_VEL
LIN {X 0,Y 502.771,Z 140.856,A -85,B 0,C 180,E1 -5783.042,E2 -5783.042} C_VEL
LIN {X 0,Y 502.767,Z 140.858,A -85,B 0,C 180,E1 -5785.68,E2 -5785.68} C_VEL
LIN {X 0,Y 502.751,Z 140.855,A -85,B 0,C 180,E1 -5788.378,E2 -5788.378} C_VEL
LIN {X 0,Y 502.763,Z 140.859,A -85,B 0,C 180,E1 -5791.495,E2 -5791.495} C_VEL
LIN {X 0,Y 502.778,Z 140.852,A -85,B 0,C 180,E1 -5794.441,E2 -5794.441} C_VEL
LIN {X 0,Y 502.729,Z 140.867,A -85,B 0,C 180,E1 -5797.172,E2 -5797.172} C_VEL
LIN {X 0,Y 502.762,Z 140.854,A -85,B 0,C 180,E1 -5800.018,E2 -5800.018} C_VEL
LIN {X 0,Y 502.733,Z 140.863,A -85,B 0,C 180,E1 -5803.236,E2 -5803.236} C_VEL
LIN {X 0,Y 502.761,Z 140.855,A -85,B 0,C 180,E1 -5805.659,E2 -5805.659} C_VEL
LIN {X 0,Y 502.756,Z 140.862,A -85,B 0,C 180,E1 -5809.013,E2 -5809.013} C_VEL
LIN {X 0,Y 502.754,Z 140.855,A -85,B 0,C 180,E1 -5812.044,E2 -5812.044} C_VEL
LIN {X 0,Y 502.777,Z 140.857,A -85,B 0,C 180,E1 -5815.033,E2 -5815.033} C_VEL
LIN {X 0,Y 502.754,Z 140.855,A -85,B 0,C 180,E1 -5817.914,E2 -5817.914} C_VEL
LIN {X 0,Y 502.749,Z 140.863,A -85,B 0,C 180,E1 -5820.708,E2 -5820.708} C_VEL
LIN {X 0,Y 502.769,Z 140.857,A -85,B 0,C 180,E1 -5823.461,E2 -5823.461} C_VEL
LIN {X 0,Y 502.775,Z 140.901,A -85,B 0,C 180,E1 -5825.312,E2 -5825.312} C_VEL
LIN {X 0,Y 504.46,Z 150.485,A -85,B 0,C 180,E1 -5827.041,E2 -5827.041} C_VEL
LIN {X 0,Y 504.066,Z 165.68,A -85,B 0,C 180,E1 -5829.601,E2 -5829.601} C_VEL
LIN {X 0,Y 503.587,Z 180.845,A -85,B 0,C 180,E1 -5832.121,E2 -5832.121} C_VEL
LIN {X 0,Y 503.257,Z 193.529,A -85,B 0,C 180,E1 -5834.205,E2 -5834.205} C_VEL
LIN {X 0,Y 505.275,Z 207.711,A -85,B 0,C 180,E1 -5834.486,E2 -5834.486} C_VEL
LIN {X 0,Y 504.733,Z 301.779,A -85,B 0,C 180,E1 -5835.897,E2 -5835.897} C_VEL
LIN {X 0,Y 504.451,Z 314.899,A -85,B 0,C 180,E1 -5836.249,E2 -5836.249} C_VEL
LIN {X 0,Y 504.149,Z 327.585,A -85,B 0,C 180,E1 -5836.754,E2 -5836.754} C_VEL
LIN {X 0,Y 503.809,Z 339.065,A -85,B 0,C 180,E1 -5837.371,E2 -5837.371} C_VEL
LIN {X 0,Y 503.486,Z 351.227,A -85,B 0,C 180,E1 -5838.221,E2 -5838.221} C_VEL
LIN {X 0,Y 503.164,Z 361.633,A -85,B 0,C 180,E1 -5839.132,E2 -5839.132} C_VEL
LIN {X 0,Y 502.805,Z 370.972,A -85,B 0,C 180,E1 -5840.142,E2 -5840.142} C_VEL
LIN {X 0,Y 502.551,Z 380.029,A -85,B 0,C 180,E1 -5841.354,E2 -5841.354} C_VEL
LIN {X 0,Y 502.342,Z 387.322,A -85,B 0,C 180,E1 -5842.565,E2 -5842.565} C_VEL
LIN {X 0,Y 502.234,Z 392.245,A -85,B 0,C 180,E1 -5843.573,E2 -5843.573} C_VEL
LIN {X 0,Y 502.171,Z 397.025,A -85,B 0,C 180,E1 -5844.781,E2 -5844.781} C_VEL
LIN {X 0,Y 502.137,Z 400.676,A -85,B 0,C 180,E1 -5845.988,E2 -5845.988} C_VEL
LIN {X 0,Y 502.12,Z 402.559,A -85,B 0,C 180,E1 -5846.791,E2 -5846.791} C_VEL
LIN {X 0,Y 502.092,Z 403.97,A -85,B 0,C 180,E1 -5847.594,E2 -5847.594} C_VEL
LIN {X 0,Y 501.992,Z 405.581,A -85,B 0,C 180,E1 -5849.199,E2 -5849.199} C_VEL
LIN {X 0,Y 501.984,Z 405.795,A -85,B 0,C 180,E1 -5850.001,E2 -5850.001} C_VEL
LIN {X 0,Y 501.993,Z 405.571,A -85,B 0,C 180,E1 -5850.803,E2 -5850.803} C_VEL
LIN {X 0,Y 502.092,Z 403.936,A -85,B 0,C 180,E1 -5852.407,E2 -5852.407} C_VEL
LIN {X 0,Y 502.12,Z 402.513,A -85,B 0,C 180,E1 -5853.21,E2 -5853.21} C_VEL
LIN {X 0,Y 502.1,Z 399.526,A -85,B 0,C 180,E1 -5854.416,E2 -5854.416} C_VEL
LIN {X 0,Y 502.199,Z 395.487,A -85,B 0,C 180,E1 -5855.622,E2 -5855.622} C_VEL
LIN {X 0,Y 502.33,Z 389.366,A -85,B 0,C 180,E1 -5857.012,E2 -5857.012} C_VEL
LIN {X 0,Y 502.448,Z 382.469,A -85,B 0,C 180,E1 -5858.244,E2 -5858.244} C_VEL
LIN {X 0,Y 502.69,Z 374.036,A -85,B 0,C 180,E1 -5859.456,E2 -5859.456} C_VEL
LIN {X 0,Y 502.95,Z 365.343,A -85,B 0,C 180,E1 -5860.467,E2 -5860.467} C_VEL
LIN {X 0,Y 503.33,Z 354.631,A -85,B 0,C 180,E1 -5861.478,E2 -5861.478} C_VEL
LIN {X 0,Y 503.606,Z 344.269,A -85,B 0,C 180,E1 -5862.269,E2 -5862.269} C_VEL
LIN {X 0,Y 504.006,Z 332.185,A -85,B 0,C 180,E1 -5862.995,E2 -5862.995} C_VEL
LIN {X 0,Y 504.292,Z 319.919,A -85,B 0,C 180,E1 -5863.551,E2 -5863.551} C_VEL
LIN {X 0,Y 504.588,Z 306.547,A -85,B 0,C 180,E1 -5863.98,E2 -5863.98} C_VEL
LIN {X 0,Y 504.809,Z 291.614,A -85,B 0,C 180,E1 -5864.256,E2 -5864.256} C_VEL
LIN {X 0,Y 505.165,Z 205.913,A -85,B 0,C 180,E1 -5865.543,E2 -5865.543} C_VEL
LIN {X 0,Y 503.203,Z 192.921,A -85,B 0,C 180,E1 -5865.818,E2 -5865.818} C_VEL
LIN {X 0,Y 503.703,Z 173.701,A -85,B 0,C 180,E1 -5868.93,E2 -5868.93} C_VEL
LIN {X 0,Y 504.112,Z 156.886,A -85,B 0,C 180,E1 -5871.682,E2 -5871.682} C_VEL
LIN {X 0,Y 504.176,Z 148.504,A -85,B 0,C 180,E1 -5873.072,E2 -5873.072} C_VEL
LIN {X 0,Y 502.787,Z 140.857,A -85,B 0,C 180,E1 -5874.444,E2 -5874.444} C_VEL
LIN {X 0,Y 502.771,Z 140.863,A -85,B 0,C 180,E1 -5877.471,E2 -5877.471} C_VEL
LIN {X 0,Y 502.745,Z 140.858,A -85,B 0,C 180,E1 -5880.216,E2 -5880.216} C_VEL
LIN {X 0,Y 502.801,Z 140.857,A -85,B 0,C 180,E1 -5883.034,E2 -5883.034} C_VEL
LIN {X 0,Y 502.749,Z 140.857,A -85,B 0,C 180,E1 -5885.954,E2 -5885.954} C_VEL
LIN {X 0,Y 502.784,Z 140.86,A -85,B 0,C 180,E1 -5888.978,E2 -5888.978} C_VEL
LIN {X 0,Y 502.747,Z 140.857,A -85,B 0,C 180,E1 -5892.192,E2 -5892.192} C_VEL
LIN {X 0,Y 502.788,Z 140.851,A -85,B 0,C 180,E1 -5895.47,E2 -5895.47} C_VEL
LIN {X 0,Y 502.764,Z 140.858,A -85,B 0,C 180,E1 -5898.928,E2 -5898.928} C_VEL
LIN {X 0,Y 502.774,Z 140.853,A -85,B 0,C 180,E1 -5902.044,E2 -5902.044} C_VEL
LIN {X 0,Y 502.791,Z 140.854,A -85,B 0,C 180,E1 -5905.034,E2 -5905.034} C_VEL
LIN {X 0,Y 502.781,Z 140.854,A -85,B 0,C 180,E1 -5907.915,E2 -5907.915} C_VEL
LIN {X 0,Y 502.792,Z 140.854,A -85,B 0,C 180,E1 -5910.71,E2 -5910.71} C_VEL
LIN {X 0,Y 502.777,Z 140.853,A -85,B 0,C 180,E1 -5913.46,E2 -5913.46} C_VEL
LIN {X 0,Y 502.77,Z 140.859,A -85,B 0,C 180,E1 -5916.085,E2 -5916.085} C_VEL
LIN {X 0,Y 502.781,Z 140.853,A -85,B 0,C 180,E1 -5918.689,E2 -5918.689} C_VEL
LIN {X 0,Y 502.81,Z 140.849,A -85,B 0,C 180,E1 -5921.248,E2 -5921.248} C_VEL
LIN {X 0,Y 502.84,Z 140.847,A -85,B 0,C 180,E1 -5924.665,E2 -5924.665} C_VEL
LIN {X 0,Y 502.881,Z 140.847,A -85,B 0,C 180,E1 -5928.039,E2 -5928.039} C_VEL
LIN {X 0,Y 502.853,Z 140.846,A -85,B 0,C 180,E1 -5931.156,E2 -5931.156} C_VEL
LIN {X 0,Y 502.873,Z 140.848,A -85,B 0,C 180,E1 -5933.581,E2 -5933.581} C_VEL
LIN {X 0,Y 502.839,Z 140.846,A -85,B 0,C 180,E1 -5936.795,E2 -5936.795} C_VEL
LIN {X 0,Y 502.897,Z 140.84,A -85,B 0,C 180,E1 -5938.399,E2 -5938.399} C_VEL
LIN {X 0,Y 503.01,Z 140.831,A -85,B 0,C 180,E1 -5940,E2 -5940} C_VEL
LIN {X 0,Y 503.021,Z 140.826,A -85,B 0,C 180,E1 -5942.402,E2 -5942.402} C_VEL
LIN {X 0,Y 502.92,Z 140.843,A -85,B 0,C 180,E1 -5945.614,E2 -5945.614} C_VEL
LIN {X 0,Y 502.913,Z 140.926,A -85,B 0,C 180,E1 -5947.402,E2 -5947.402} C_VEL
LIN {X 0,Y 503.582,Z 146.456,A -85,B 0,C 180,E1 -5948.427,E2 -5948.427} C_VEL
LIN {X 0,Y 503.428,Z 161.071,A -85,B 0,C 180,E1 -5951.067,E2 -5951.067} C_VEL
LIN {X 0,Y 503.371,Z 167.897,A -85,B 0,C 180,E1 -5952.26,E2 -5952.26} C_VEL
LIN {X 0,Y 505.456,Z 180.308,A -85,B 0,C 180,E1 -5952.523,E2 -5952.523} C_VEL
LIN {X 0,Y 504.728,Z 275.816,A -85,B 0,C 180,E1 -5953.975,E2 -5953.975} C_VEL
LIN {X 0,Y 504.5,Z 289.001,A -85,B 0,C 180,E1 -5954.342,E2 -5954.342} C_VEL
LIN {X 0,Y 504.269,Z 301.168,A -85,B 0,C 180,E1 -5954.839,E2 -5954.839} C_VEL
LIN {X 0,Y 503.967,Z 312.574,A -85,B 0,C 180,E1 -5955.463,E2 -5955.463} C_VEL
LIN {X 0,Y 503.569,Z 324.62,A -85,B 0,C 180,E1 -5956.313,E2 -5956.313} C_VEL
LIN {X 0,Y 503.225,Z 335.304,A -85,B 0,C 180,E1 -5957.264,E2 -5957.264} C_VEL
LIN {X 0,Y 502.972,Z 343.536,A -85,B 0,C 180,E1 -5958.164,E2 -5958.164} C_VEL
LIN {X 0,Y 502.656,Z 352.7,A -85,B 0,C 180,E1 -5959.395,E2 -5959.395} C_VEL
LIN {X 0,Y 502.44,Z 360.372,A -85,B 0,C 180,E1 -5960.683,E2 -5960.683} C_VEL
LIN {X 0,Y 502.332,Z 365.509,A -85,B 0,C 180,E1 -5961.763,E2 -5961.763} C_VEL
LIN {X 0,Y 502.194,Z 370.431,A -85,B 0,C 180,E1 -5963.07,E2 -5963.07} C_VEL
LIN {X 0,Y 502.096,Z 374.381,A -85,B 0,C 180,E1 -5964.518,E2 -5964.518} C_VEL
LIN {X 0,Y 502.006,Z 376.597,A -85,B 0,C 180,E1 -5965.722,E2 -5965.722} C_VEL
LIN {X 0,Y 502.001,Z 377.644,A -85,B 0,C 180,E1 -5966.616,E2 -5966.616} C_VEL
LIN {X 0,Y 501.988,Z 378.277,A -85,B 0,C 180,E1 -5968.112,E2 -5968.112} C_VEL
LIN {X 0,Y 502.038,Z 377.312,A -85,B 0,C 180,E1 -5969.78,E2 -5969.78} C_VEL
LIN {X 0,Y 502.146,Z 374.762,A -85,B 0,C 180,E1 -5971.377,E2 -5971.377} C_VEL
LIN {X 0,Y 502.164,Z 370.773,A -85,B 0,C 180,E1 -5972.888,E2 -5972.888} C_VEL
LIN {X 0,Y 502.289,Z 365.296,A -85,B 0,C 180,E1 -5974.357,E2 -5974.357} C_VEL
LIN {X 0,Y 502.48,Z 358.199,A -85,B 0,C 180,E1 -5975.784,E2 -5975.784} C_VEL
LIN {X 0,Y 502.75,Z 350.884,A -85,B 0,C 180,E1 -5976.949,E2 -5976.949} C_VEL
LIN {X 0,Y 502.768,Z 350.094,A -85,B 0,C 180,E1 -5977.059,E2 -5977.059} C_VEL
LIN {X 0,Y 502.202,Z 346.364,A -85,B 0,C 180,E1 -5977.576,E2 -5977.576} C_VEL
LIN {X 0,Y 499.521,Z 340.016,A -85,B 0,C 180,E1 -5978.399,E2 -5978.399} C_VEL
LIN {X 0,Y 496.9,Z 333.194,A -85,B 0,C 180,E1 -5979.17,E2 -5979.17} C_VEL
LIN {X 0,Y 496.42,Z 328.646,A -85,B 0,C 180,E1 -5979.6,E2 -5979.6} C_VEL
LIN {X 0,Y 496.802,Z 317.606,A -85,B 0,C 180,E1 -5980.468,E2 -5980.468} C_VEL
LIN {X 0,Y 497.202,Z 306.46,A -85,B 0,C 180,E1 -5981.161,E2 -5981.161} C_VEL
LIN {X 0,Y 497.478,Z 294.218,A -85,B 0,C 180,E1 -5981.74,E2 -5981.74} C_VEL
LIN {X 0,Y 497.748,Z 280.846,A -85,B 0,C 180,E1 -5982.188,E2 -5982.188} C_VEL
LIN {X 0,Y 497.936,Z 267.474,A -85,B 0,C 180,E1 -5982.459,E2 -5982.459} C_VEL
LIN {X 0,Y 498.451,Z 179.408,A -85,B 0,C 180,E1 -5983.793,E2 -5983.793} C_VEL
LIN {X 0,Y 496.297,Z 167.685,A -85,B 0,C 180,E1 -5984.057,E2 -5984.057} C_VEL
LIN {X 0,Y 496.789,Z 151.53,A -85,B 0,C 180,E1 -5987.23,E2 -5987.23} C_VEL
LIN {X 0,Y 496.6,Z 146.203,A -85,B 0,C 180,E1 -5988.305,E2 -5988.305} C_VEL
LIN {X 0,Y 495.78,Z 141.73,A -85,B 0,C 180,E1 -5989.272,E2 -5989.272} C_VEL
LIN {X 0,Y 495.718,Z 141.739,A -85,B 0,C 180,E1 -5992.437,E2 -5992.437} C_VEL
LIN {X 0,Y 495.771,Z 141.725,A -85,B 0,C 180,E1 -5995.456,E2 -5995.456} C_VEL
LIN {X 0,Y 495.755,Z 141.734,A -85,B 0,C 180,E1 -5998.363,E2 -5998.363} C_VEL
LIN {X 0,Y 495.732,Z 141.73,A -85,B 0,C 180,E1 -6001.52,E2 -6001.52} C_VEL
LIN {X 0,Y 495.717,Z 141.734,A -85,B 0,C 180,E1 -6003.927,E2 -6003.927} C_VEL
LIN {X 0,Y 495.749,Z 141.728,A -85,B 0,C 180,E1 -6007.144,E2 -6007.144} C_VEL
LIN {X 0,Y 495.726,Z 141.737,A -85,B 0,C 180,E1 -6010.107,E2 -6010.107} C_VEL
LIN {X 0,Y 495.707,Z 141.735,A -85,B 0,C 180,E1 -6012.678,E2 -6012.678} C_VEL
LIN {X 0,Y 495.781,Z 141.724,A -85,B 0,C 180,E1 -6015.216,E2 -6015.216} C_VEL
LIN {X 0,Y 495.827,Z 141.72,A -85,B 0,C 180,E1 -6018.554,E2 -6018.554} C_VEL
LIN {X 0,Y 495.815,Z 141.726,A -85,B 0,C 180,E1 -6021.85,E2 -6021.85} C_VEL
LIN {X 0,Y 495.855,Z 141.718,A -85,B 0,C 180,E1 -6024.305,E2 -6024.305} C_VEL
LIN {X 0,Y 495.979,Z 141.703,A -85,B 0,C 180,E1 -6027.563,E2 -6027.563} C_VEL
LIN {X 0,Y 495.976,Z 141.705,A -85,B 0,C 180,E1 -6029.999,E2 -6029.999} C_VEL
LIN {X 0,Y 495.979,Z 141.7,A -85,B 0,C 180,E1 -6032.436,E2 -6032.436} C_VEL
LIN {X 0,Y 495.848,Z 141.724,A -85,B 0,C 180,E1 -6035.693,E2 -6035.693} C_VEL
LIN {X 0,Y 495.814,Z 141.722,A -85,B 0,C 180,E1 -6038.148,E2 -6038.148} C_VEL
LIN {X 0,Y 495.824,Z 141.725,A -85,B 0,C 180,E1 -6041.445,E2 -6041.445} C_VEL
LIN {X 0,Y 495.776,Z 141.725,A -85,B 0,C 180,E1 -6044.782,E2 -6044.782} C_VEL
LIN {X 0,Y 495.749,Z 141.728,A -85,B 0,C 180,E1 -6048.225,E2 -6048.225} C_VEL
LIN {X 0,Y 495.747,Z 141.729,A -85,B 0,C 180,E1 -6050.757,E2 -6050.757} C_VEL
LIN {X 0,Y 495.735,Z 141.737,A -85,B 0,C 180,E1 -6053.387,E2 -6053.387} C_VEL
LIN {X 0,Y 495.716,Z 141.732,A -85,B 0,C 180,E1 -6056.071,E2 -6056.071} C_VEL
LIN {X 0,Y 495.718,Z 141.735,A -85,B 0,C 180,E1 -6058.817,E2 -6058.817} C_VEL
LIN {X 0,Y 495.737,Z 141.731,A -85,B 0,C 180,E1 -6061.721,E2 -6061.721} C_VEL
LIN {X 0,Y 495.756,Z 141.73,A -85,B 0,C 180,E1 -6064.691,E2 -6064.691} C_VEL
LIN {X 0,Y 495.717,Z 141.733,A -85,B 0,C 180,E1 -6067.562,E2 -6067.562} C_VEL
LIN {X 0,Y 495.74,Z 141.729,A -85,B 0,C 180,E1 -6070.044,E2 -6070.044} C_VEL
LIN {X 0,Y 495.692,Z 141.743,A -85,B 0,C 180,E1 -6072.886,E2 -6072.886} C_VEL
LIN {X 0,Y 495.718,Z 141.731,A -85,B 0,C 180,E1 -6075.997,E2 -6075.997} C_VEL
LIN {X 0,Y 495.721,Z 141.733,A -85,B 0,C 180,E1 -6079.295,E2 -6079.295} C_VEL
LIN {X 0,Y 495.722,Z 141.732,A -85,B 0,C 180,E1 -6081.405,E2 -6081.405} C_VEL
LIN {X 0,Y 495.734,Z 141.735,A -85,B 0,C 180,E1 -6084.461,E2 -6084.461} C_VEL
LIN {X 0,Y 495.745,Z 141.728,A -85,B 0,C 180,E1 -6087.404,E2 -6087.404} C_VEL
LIN {X 0,Y 495.734,Z 141.734,A -85,B 0,C 180,E1 -6090.251,E2 -6090.251} C_VEL
LIN {X 0,Y 495.732,Z 141.73,A -85,B 0,C 180,E1 -6093.27,E2 -6093.27} C_VEL
LIN {X 0,Y 495.702,Z 141.734,A -85,B 0,C 180,E1 -6095.722,E2 -6095.722} C_VEL
LIN {X 0,Y 495.725,Z 141.739,A -85,B 0,C 180,E1 -6098.37,E2 -6098.37} C_VEL
LIN {X 0,Y 495.757,Z 141.728,A -85,B 0,C 180,E1 -6100.97,E2 -6100.97} C_VEL
LIN {X 0,Y 495.795,Z 141.726,A -85,B 0,C 180,E1 -6104.557,E2 -6104.557} C_VEL
LIN {X 0,Y 495.815,Z 141.725,A -85,B 0,C 180,E1 -6107.969,E2 -6107.969} C_VEL
LIN {X 0,Y 495.786,Z 141.723,A -85,B 0,C 180,E1 -6111.029,E2 -6111.029} C_VEL
LIN {X 0,Y 495.814,Z 141.721,A -85,B 0,C 180,E1 -6113.489,E2 -6113.489} C_VEL
LIN {X 0,Y 495.697,Z 141.741,A -85,B 0,C 180,E1 -6115.935,E2 -6115.935} C_VEL
LIN {X 0,Y 495.968,Z 141.703,A -85,B 0,C 180,E1 -6117.563,E2 -6117.563} C_VEL
LIN {X 0,Y 495.964,Z 141.709,A -85,B 0,C 180,E1 -6120,E2 -6120} C_VEL
LIN {X 0,Y 495.967,Z 141.702,A -85,B 0,C 180,E1 -6122.436,E2 -6122.436} C_VEL
LIN {X 0,Y 495.842,Z 141.723,A -85,B 0,C 180,E1 -6125.694,E2 -6125.694} C_VEL
LIN {X 0,Y 495.802,Z 141.724,A -85,B 0,C 180,E1 -6128.149,E2 -6128.149} C_VEL
LIN {X 0,Y 495.813,Z 141.724,A -85,B 0,C 180,E1 -6131.446,E2 -6131.446} C_VEL
LIN {X 0,Y 495.766,Z 141.725,A -85,B 0,C 180,E1 -6134.783,E2 -6134.783} C_VEL
LIN {X 0,Y 495.739,Z 141.73,A -85,B 0,C 180,E1 -6138.226,E2 -6138.226} C_VEL
LIN {X 0,Y 495.738,Z 141.729,A -85,B 0,C 180,E1 -6140.758,E2 -6140.758} C_VEL
LIN {X 0,Y 495.722,Z 141.739,A -85,B 0,C 180,E1 -6143.388,E2 -6143.388} C_VEL
LIN {X 0,Y 495.73,Z 141.731,A -85,B 0,C 180,E1 -6146.73,E2 -6146.73} C_VEL
LIN {X 0,Y 495.687,Z 141.738,A -85,B 0,C 180,E1 -6149.752,E2 -6149.752} C_VEL
LIN {X 0,Y 495.741,Z 141.729,A -85,B 0,C 180,E1 -6152.596,E2 -6152.596} C_VEL
LIN {X 0,Y 495.722,Z 141.735,A -85,B 0,C 180,E1 -6155.54,E2 -6155.54} C_VEL
LIN {X 0,Y 495.731,Z 141.733,A -85,B 0,C 180,E1 -6158.765,E2 -6158.765} C_VEL
LIN {X 0,Y 495.717,Z 141.732,A -85,B 0,C 180,E1 -6161.785,E2 -6161.785} C_VEL
LIN {X 0,Y 495.725,Z 141.737,A -85,B 0,C 180,E1 -6165.142,E2 -6165.142} C_VEL
LIN {X 0,Y 495.717,Z 141.732,A -85,B 0,C 180,E1 -6168.216,E2 -6168.216} C_VEL
LIN {X 0,Y 495.732,Z 141.733,A -85,B 0,C 180,E1 -6171.236,E2 -6171.236} C_VEL
LIN {X 0,Y 495.723,Z 141.734,A -85,B 0,C 180,E1 -6174.461,E2 -6174.461} C_VEL
LIN {X 0,Y 495.736,Z 141.73,A -85,B 0,C 180,E1 -6177.404,E2 -6177.404} C_VEL
LIN {X 0,Y 495.692,Z 141.738,A -85,B 0,C 180,E1 -6180.25,E2 -6180.25} C_VEL
LIN {X 0,Y 495.734,Z 141.734,A -85,B 0,C 180,E1 -6183.272,E2 -6183.272} C_VEL
LIN {X 0,Y 495.731,Z 141.841,A -85,B 0,C 180,E1 -6185.139,E2 -6185.139} C_VEL
LIN {X 0,Y 497.47,Z 151.067,A -85,B 0,C 180,E1 -6186.834,E2 -6186.834} C_VEL
LIN {X 0,Y 497.254,Z 163.69,A -85,B 0,C 180,E1 -6189.002,E2 -6189.002} C_VEL
LIN {X 0,Y 496.608,Z 180.665,A -85,B 0,C 180,E1 -6191.861,E2 -6191.861} C_VEL
LIN {X 0,Y 496.267,Z 193.356,A -85,B 0,C 180,E1 -6193.98,E2 -6193.98} C_VEL
LIN {X 0,Y 498.429,Z 208.607,A -85,B 0,C 180,E1 -6194.288,E2 -6194.288} C_VEL
LIN {X 0,Y 497.818,Z 302.229,A -85,B 0,C 180,E1 -6195.723,E2 -6195.723} C_VEL
LIN {X 0,Y 497.519,Z 315.887,A -85,B 0,C 180,E1 -6196.106,E2 -6196.106} C_VEL
LIN {X 0,Y 497.198,Z 328.239,A -85,B 0,C 180,E1 -6196.617,E2 -6196.617} C_VEL
LIN {X 0,Y 496.813,Z 339.578,A -85,B 0,C 180,E1 -6197.248,E2 -6197.248} C_VEL
LIN {X 0,Y 496.493,Z 350.892,A -85,B 0,C 180,E1 -6198.053,E2 -6198.053} C_VEL
LIN {X 0,Y 496.155,Z 361.329,A -85,B 0,C 180,E1 -6198.976,E2 -6198.976} C_VEL
LIN {X 0,Y 495.773,Z 370.702,A -85,B 0,C 180,E1 -6200,E2 -6200} C_VEL
LIN {X 0,Y 495.473,Z 379.778,A -85,B 0,C 180,E1 -6201.23,E2 -6201.23} C_VEL
LIN {X 0,Y 495.273,Z 387.089,A -85,B 0,C 180,E1 -6202.458,E2 -6202.458} C_VEL
LIN {X 0,Y 495.117,Z 393.26,A -85,B 0,C 180,E1 -6203.766,E2 -6203.766} C_VEL
LIN {X 0,Y 495.033,Z 398.149,A -85,B 0,C 180,E1 -6205.114,E2 -6205.114} C_VEL
LIN {X 0,Y 495.03,Z 400.472,A -85,B 0,C 180,E1 -6205.93,E2 -6205.93} C_VEL
LIN {X 0,Y 495.041,Z 402.36,A -85,B 0,C 180,E1 -6206.745,E2 -6206.745} C_VEL
LIN {X 0,Y 494.998,Z 403.774,A -85,B 0,C 180,E1 -6207.56,E2 -6207.56} C_VEL
LIN {X 0,Y 494.962,Z 404.777,A -85,B 0,C 180,E1 -6208.373,E2 -6208.373} C_VEL
LIN {X 0,Y 494.902,Z 405.601,A -85,B 0,C 180,E1 -6210.001,E2 -6210.001} C_VEL
LIN {X 0,Y 494.913,Z 405.375,A -85,B 0,C 180,E1 -6210.814,E2 -6210.814} C_VEL
LIN {X 0,Y 494.962,Z 404.752,A -85,B 0,C 180,E1 -6211.628,E2 -6211.628} C_VEL
LIN {X 0,Y 494.998,Z 403.735,A -85,B 0,C 180,E1 -6212.442,E2 -6212.442} C_VEL
LIN {X 0,Y 495.042,Z 402.308,A -85,B 0,C 180,E1 -6213.256,E2 -6213.256} C_VEL
LIN {X 0,Y 495.006,Z 399.314,A -85,B 0,C 180,E1 -6214.479,E2 -6214.479} C_VEL
LIN {X 0,Y 495.115,Z 395.265,A -85,B 0,C 180,E1 -6215.703,E2 -6215.703} C_VEL
LIN {X 0,Y 495.254,Z 389.028,A -85,B 0,C 180,E1 -6217.133,E2 -6217.133} C_VEL
LIN {X 0,Y 495.406,Z 382.22,A -85,B 0,C 180,E1 -6218.362,E2 -6218.362} C_VEL
LIN {X 0,Y 495.651,Z 373.766,A -85,B 0,C 180,E1 -6219.591,E2 -6219.591} C_VEL
LIN {X 0,Y 495.956,Z 365.05,A -85,B 0,C 180,E1 -6220.616,E2 -6220.616} C_VEL
LIN {X 0,Y 496.337,Z 354.319,A -85,B 0,C 180,E1 -6221.641,E2 -6221.641} C_VEL
LIN {X 0,Y 496.642,Z 343.629,A -85,B 0,C 180,E1 -6222.466,E2 -6222.466} C_VEL
LIN {X 0,Y 497.052,Z 331.825,A -85,B 0,C 180,E1 -6223.18,E2 -6223.18} C_VEL
LIN {X 0,Y 497.404,Z 318.235,A -85,B 0,C 180,E1 -6223.795,E2 -6223.795} C_VEL
LIN {X 0,Y 497.73,Z 305.009,A -85,B 0,C 180,E1 -6224.202,E2 -6224.202} C_VEL
LIN {X 0,Y 497.942,Z 287.612,A -85,B 0,C 180,E1 -6224.509,E2 -6224.509} C_VEL
LIN {X 0,Y 498.399,Z 207.042,A -85,B 0,C 180,E1 -6225.744,E2 -6225.744} C_VEL
LIN {X 0,Y 496.216,Z 192.742,A -85,B 0,C 180,E1 -6226.047,E2 -6226.047} C_VEL
LIN {X 0,Y 496.737,Z 173.52,A -85,B 0,C 180,E1 -6229.206,E2 -6229.206} C_VEL
LIN {X 0,Y 497.198,Z 156.694,A -85,B 0,C 180,E1 -6231.999,E2 -6231.999} C_VEL
LIN {X 0,Y 497.29,Z 150.125,A -85,B 0,C 180,E1 -6233.105,E2 -6233.105} C_VEL
LIN {X 0,Y 495.729,Z 141.737,A -85,B 0,C 180,E1 -6234.623,E2 -6234.623} C_VEL
LIN {X 0,Y 495.711,Z 141.738,A -85,B 0,C 180,E1 -6237.896,E2 -6237.896} C_VEL
LIN {X 0,Y 495.711,Z 141.737,A -85,B 0,C 180,E1 -6240.691,E2 -6240.691} C_VEL
LIN {X 0,Y 495.741,Z 141.733,A -85,B 0,C 180,E1 -6243.566,E2 -6243.566} C_VEL
LIN {X 0,Y 495.694,Z 141.738,A -85,B 0,C 180,E1 -6246.548,E2 -6246.548} C_VEL
LIN {X 0,Y 495.744,Z 141.731,A -85,B 0,C 180,E1 -6249.64,E2 -6249.64} C_VEL
LIN {X 0,Y 495.697,Z 141.741,A -85,B 0,C 180,E1 -6252.887,E2 -6252.887} C_VEL
LIN {X 0,Y 495.725,Z 141.73,A -85,B 0,C 180,E1 -6255.998,E2 -6255.998} C_VEL
LIN {X 0,Y 495.728,Z 141.731,A -85,B 0,C 180,E1 -6259.296,E2 -6259.296} C_VEL
LIN {X 0,Y 495.73,Z 141.729,A -85,B 0,C 180,E1 -6261.406,E2 -6261.406} C_VEL
LIN {X 0,Y 495.742,Z 141.733,A -85,B 0,C 180,E1 -6264.462,E2 -6264.462} C_VEL
LIN {X 0,Y 495.753,Z 141.728,A -85,B 0,C 180,E1 -6267.405,E2 -6267.405} C_VEL
LIN {X 0,Y 495.743,Z 141.733,A -85,B 0,C 180,E1 -6270.252,E2 -6270.252} C_VEL
LIN {X 0,Y 495.741,Z 141.729,A -85,B 0,C 180,E1 -6273.271,E2 -6273.271} C_VEL
LIN {X 0,Y 495.742,Z 141.732,A -85,B 0,C 180,E1 -6276.612,E2 -6276.612} C_VEL
LIN {X 0,Y 495.783,Z 141.722,A -85,B 0,C 180,E1 -6279.324,E2 -6279.324} C_VEL
LIN {X 0,Y 495.783,Z 141.728,A -85,B 0,C 180,E1 -6281.829,E2 -6281.829} C_VEL
LIN {X 0,Y 495.785,Z 141.725,A -85,B 0,C 180,E1 -6285.217,E2 -6285.217} C_VEL
LIN {X 0,Y 495.854,Z 141.718,A -85,B 0,C 180,E1 -6288.555,E2 -6288.555} C_VEL
LIN {X 0,Y 495.817,Z 141.728,A -85,B 0,C 180,E1 -6291.851,E2 -6291.851} C_VEL
LIN {X 0,Y 495.859,Z 141.718,A -85,B 0,C 180,E1 -6294.306,E2 -6294.306} C_VEL
LIN {X 0,Y 495.981,Z 141.707,A -85,B 0,C 180,E1 -6297.564,E2 -6297.564} C_VEL
LIN {X 0,Y 495.979,Z 141.707,A -85,B 0,C 180,E1 -6300,E2 -6300} C_VEL
LIN {X 0,Y 495.989,Z 141.703,A -85,B 0,C 180,E1 -6302.437,E2 -6302.437} C_VEL
LIN {X 0,Y 495.876,Z 141.72,A -85,B 0,C 180,E1 -6305.694,E2 -6305.694} C_VEL
LIN {X 0,Y 495.892,Z 141.777,A -85,B 0,C 180,E1 -6307.235,E2 -6307.235} C_VEL
LIN {X 0,Y 496.637,Z 147.631,A -85,B 0,C 180,E1 -6308.34,E2 -6308.34} C_VEL
LIN {X 0,Y 496.445,Z 162.351,A -85,B 0,C 180,E1 -6311.018,E2 -6311.018} C_VEL
LIN {X 0,Y 496.378,Z 167.947,A -85,B 0,C 180,E1 -6312.019,E2 -6312.019} C_VEL
LIN {X 0,Y 498.614,Z 180.035,A -85,B 0,C 180,E1 -6312.289,E2 -6312.289} C_VEL
LIN {X 0,Y 497.837,Z 276.054,A -85,B 0,C 180,E1 -6313.783,E2 -6313.783} C_VEL
LIN {X 0,Y 497.602,Z 289.191,A -85,B 0,C 180,E1 -6314.154,E2 -6314.154} C_VEL
LIN {X 0,Y 497.331,Z 301.917,A -85,B 0,C 180,E1 -6314.684,E2 -6314.684} C_VEL
LIN {X 0,Y 496.992,Z 314.088,A -85,B 0,C 180,E1 -6315.376,E2 -6315.376} C_VEL
LIN {X 0,Y 496.606,Z 325.097,A -85,B 0,C 180,E1 -6316.175,E2 -6316.175} C_VEL
LIN {X 0,Y 496.254,Z 335.232,A -85,B 0,C 180,E1 -6317.09,E2 -6317.09} C_VEL
LIN {X 0,Y 495.909,Z 344.828,A -85,B 0,C 180,E1 -6318.167,E2 -6318.167} C_VEL
LIN {X 0,Y 495.639,Z 352.712,A -85,B 0,C 180,E1 -6319.25,E2 -6319.25} C_VEL
LIN {X 0,Y 495.383,Z 360.412,A -85,B 0,C 180,E1 -6320.553,E2 -6320.553} C_VEL
LIN {X 0,Y 495.271,Z 365.591,A -85,B 0,C 180,E1 -6321.651,E2 -6321.651} C_VEL
LIN {X 0,Y 495.106,Z 370.661,A -85,B 0,C 180,E1 -6323.012,E2 -6323.012} C_VEL
LIN {X 0,Y 495.017,Z 374.237,A -85,B 0,C 180,E1 -6324.314,E2 -6324.314} C_VEL
LIN {X 0,Y 494.946,Z 376.043,A -85,B 0,C 180,E1 -6325.213,E2 -6325.213} C_VEL
LIN {X 0,Y 494.907,Z 377.782,A -85,B 0,C 180,E1 -6326.537,E2 -6326.537} C_VEL
LIN {X 0,Y 494.923,Z 378.43,A -85,B 0,C 180,E1 -6328.307,E2 -6328.307} C_VEL
LIN {X 0,Y 494.969,Z 377.314,A -85,B 0,C 180,E1 -6329.987,E2 -6329.987} C_VEL
LIN {X 0,Y 494.995,Z 376.233,A -85,B 0,C 180,E1 -6330.74,E2 -6330.74} C_VEL
LIN {X 0,Y 495.064,Z 373.203,A -85,B 0,C 180,E1 -6332.165,E2 -6332.165} C_VEL
LIN {X 0,Y 495.117,Z 368.73,A -85,B 0,C 180,E1 -6333.614,E2 -6333.614} C_VEL
LIN {X 0,Y 495.255,Z 363.738,A -85,B 0,C 180,E1 -6334.832,E2 -6334.832} C_VEL
LIN {X 0,Y 495.462,Z 357.494,A -85,B 0,C 180,E1 -6336.047,E2 -6336.047} C_VEL
LIN {X 0,Y 495.76,Z 349.757,A -85,B 0,C 180,E1 -6337.252,E2 -6337.252} C_VEL
LIN {X 0,Y 496.096,Z 340.376,A -85,B 0,C 180,E1 -6338.431,E2 -6338.431} C_VEL
LIN {X 0,Y 496.369,Z 330.098,A -85,B 0,C 180,E1 -6339.474,E2 -6339.474} C_VEL
LIN {X 0,Y 496.42,Z 328.646,A -85,B 0,C 180,E1 -6339.6,E2 -6339.6} C_VEL
LIN {X 0,Y 495.947,Z 323.987,A -85,B 0,C 180,E1 -6340.008,E2 -6340.008} C_VEL
LIN {X 0,Y 493.39,Z 316.231,A -85,B 0,C 180,E1 -6340.653,E2 -6340.653} C_VEL
LIN {X 0,Y 490.875,Z 308.039,A -85,B 0,C 180,E1 -6341.236,E2 -6341.236} C_VEL
LIN {X 0,Y 490.418,Z 302.691,A -85,B 0,C 180,E1 -6341.541,E2 -6341.541} C_VEL
LIN {X 0,Y 490.68,Z 290.509,A -85,B 0,C 180,E1 -6342.075,E2 -6342.075} C_VEL
LIN {X 0,Y 490.923,Z 277.598,A -85,B 0,C 180,E1 -6342.461,E2 -6342.461} C_VEL
LIN {X 0,Y 491.106,Z 257.387,A -85,B 0,C 180,E1 -6342.807,E2 -6342.807} C_VEL
LIN {X 0,Y 491.613,Z 180.168,A -85,B 0,C 180,E1 -6343.999,E2 -6343.999} C_VEL
LIN {X 0,Y 489.32,Z 167.779,A -85,B 0,C 180,E1 -6344.296,E2 -6344.296} C_VEL
LIN {X 0,Y 489.823,Z 152.582,A -85,B 0,C 180,E1 -6347.319,E2 -6347.319} C_VEL
LIN {X 0,Y 489.678,Z 147.891,A -85,B 0,C 180,E1 -6348.273,E2 -6348.273} C_VEL
LIN {X 0,Y 488.729,Z 142.608,A -85,B 0,C 180,E1 -6349.405,E2 -6349.405} C_VEL
LIN {X 0,Y 488.665,Z 142.616,A -85,B 0,C 180,E1 -6352.281,E2 -6352.281} C_VEL
LIN {X 0,Y 488.722,Z 142.605,A -85,B 0,C 180,E1 -6355.054,E2 -6355.054} C_VEL
LIN {X 0,Y 488.703,Z 142.608,A -85,B 0,C 180,E1 -6358.047,E2 -6358.047} C_VEL
LIN {X 0,Y 488.669,Z 142.609,A -85,B 0,C 180,E1 -6361.319,E2 -6361.319} C_VEL
LIN {X 0,Y 488.685,Z 142.608,A -85,B 0,C 180,E1 -6363.523,E2 -6363.523} C_VEL
LIN {X 0,Y 488.666,Z 142.618,A -85,B 0,C 180,E1 -6366.253,E2 -6366.253} C_VEL
LIN {X 0,Y 488.702,Z 142.605,A -85,B 0,C 180,E1 -6369.191,E2 -6369.191} C_VEL
LIN {X 0,Y 488.711,Z 142.606,A -85,B 0,C 180,E1 -6371.647,E2 -6371.647} C_VEL
LIN {X 0,Y 488.747,Z 142.6,A -85,B 0,C 180,E1 -6374.998,E2 -6374.998} C_VEL
LIN {X 0,Y 488.789,Z 142.598,A -85,B 0,C 180,E1 -6378.387,E2 -6378.387} C_VEL
LIN {X 0,Y 488.762,Z 142.603,A -85,B 0,C 180,E1 -6381.732,E2 -6381.732} C_VEL
LIN {X 0,Y 488.815,Z 142.596,A -85,B 0,C 180,E1 -6384.223,E2 -6384.223} C_VEL
LIN {X 0,Y 488.945,Z 142.579,A -85,B 0,C 180,E1 -6387.528,E2 -6387.528} C_VEL
LIN {X 0,Y 488.945,Z 142.581,A -85,B 0,C 180,E1 -6389.999,E2 -6389.999} C_VEL
LIN {X 0,Y 488.945,Z 142.576,A -85,B 0,C 180,E1 -6392.471,E2 -6392.471} C_VEL
LIN {X 0,Y 488.807,Z 142.6,A -85,B 0,C 180,E1 -6395.776,E2 -6395.776} C_VEL
LIN {X 0,Y 488.76,Z 142.599,A -85,B 0,C 180,E1 -6398.267,E2 -6398.267} C_VEL
LIN {X 0,Y 488.787,Z 142.603,A -85,B 0,C 180,E1 -6401.612,E2 -6401.612} C_VEL
LIN {X 0,Y 488.748,Z 142.602,A -85,B 0,C 180,E1 -6405,E2 -6405} C_VEL
LIN {X 0,Y 488.708,Z 142.605,A -85,B 0,C 180,E1 -6408.443,E2 -6408.443} C_VEL
LIN {X 0,Y 488.691,Z 142.611,A -85,B 0,C 180,E1 -6411.071,E2 -6411.071} C_VEL
LIN {X 0,Y 488.665,Z 142.613,A -85,B 0,C 180,E1 -6413.746,E2 -6413.746} C_VEL
LIN {X 0,Y 488.681,Z 142.608,A -85,B 0,C 180,E1 -6416.475,E2 -6416.475} C_VEL
LIN {X 0,Y 488.687,Z 142.615,A -85,B 0,C 180,E1 -6419.272,E2 -6419.272} C_VEL
LIN {X 0,Y 488.689,Z 142.607,A -85,B 0,C 180,E1 -6422.147,E2 -6422.147} C_VEL
LIN {X 0,Y 488.709,Z 142.613,A -85,B 0,C 180,E1 -6425.115,E2 -6425.115} C_VEL
LIN {X 0,Y 488.672,Z 142.609,A -85,B 0,C 180,E1 -6428.2,E2 -6428.2} C_VEL
LIN {X 0,Y 488.691,Z 142.608,A -85,B 0,C 180,E1 -6430.34,E2 -6430.34} C_VEL
LIN {X 0,Y 488.67,Z 142.61,A -85,B 0,C 180,E1 -6433.655,E2 -6433.655} C_VEL
LIN {X 0,Y 488.669,Z 142.612,A -85,B 0,C 180,E1 -6436.343,E2 -6436.343} C_VEL
LIN {X 0,Y 488.699,Z 142.606,A -85,B 0,C 180,E1 -6439.673,E2 -6439.673} C_VEL
LIN {X 0,Y 488.66,Z 142.617,A -85,B 0,C 180,E1 -6442.839,E2 -6442.839} C_VEL
LIN {X 0,Y 488.712,Z 142.605,A -85,B 0,C 180,E1 -6445.885,E2 -6445.885} C_VEL
LIN {X 0,Y 488.677,Z 142.614,A -85,B 0,C 180,E1 -6448.819,E2 -6448.819} C_VEL
LIN {X 0,Y 488.685,Z 142.608,A -85,B 0,C 180,E1 -6451.667,E2 -6451.667} C_VEL
LIN {X 0,Y 488.683,Z 142.616,A -85,B 0,C 180,E1 -6454.44,E2 -6454.44} C_VEL
LIN {X 0,Y 488.7,Z 142.606,A -85,B 0,C 180,E1 -6457.152,E2 -6457.152} C_VEL
LIN {X 0,Y 488.709,Z 142.606,A -85,B 0,C 180,E1 -6459.809,E2 -6459.809} C_VEL
LIN {X 0,Y 488.663,Z 142.617,A -85,B 0,C 180,E1 -6462.42,E2 -6462.42} C_VEL
LIN {X 0,Y 488.739,Z 142.601,A -85,B 0,C 180,E1 -6464.999,E2 -6464.999} C_VEL
LIN {X 0,Y 488.776,Z 142.602,A -85,B 0,C 180,E1 -6468.387,E2 -6468.387} C_VEL
LIN {X 0,Y 488.749,Z 142.603,A -85,B 0,C 180,E1 -6471.732,E2 -6471.732} C_VEL
LIN {X 0,Y 488.806,Z 142.599,A -85,B 0,C 180,E1 -6474.223,E2 -6474.223} C_VEL
LIN {X 0,Y 488.933,Z 142.579,A -85,B 0,C 180,E1 -6477.528,E2 -6477.528} C_VEL
LIN {X 0,Y 488.933,Z 142.584,A -85,B 0,C 180,E1 -6480,E2 -6480} C_VEL
LIN {X 0,Y 488.933,Z 142.578,A -85,B 0,C 180,E1 -6482.471,E2 -6482.471} C_VEL
LIN {X 0,Y 488.802,Z 142.601,A -85,B 0,C 180,E1 -6485.776,E2 -6485.776} C_VEL
LIN {X 0,Y 488.748,Z 142.602,A -85,B 0,C 180,E1 -6488.267,E2 -6488.267} C_VEL
LIN {X 0,Y 488.775,Z 142.604,A -85,B 0,C 180,E1 -6491.613,E2 -6491.613} C_VEL
LIN {X 0,Y 488.738,Z 142.602,A -85,B 0,C 180,E1 -6495.001,E2 -6495.001} C_VEL
LIN {X 0,Y 488.697,Z 142.606,A -85,B 0,C 180,E1 -6498.444,E2 -6498.444} C_VEL
LIN {X 0,Y 488.682,Z 142.611,A -85,B 0,C 180,E1 -6501.072,E2 -6501.072} C_VEL
LIN {X 0,Y 488.652,Z 142.616,A -85,B 0,C 180,E1 -6503.748,E2 -6503.748} C_VEL
LIN {X 0,Y 488.673,Z 142.609,A -85,B 0,C 180,E1 -6506.477,E2 -6506.477} C_VEL
LIN {X 0,Y 488.651,Z 142.62,A -85,B 0,C 180,E1 -6509.275,E2 -6509.275} C_VEL
LIN {X 0,Y 488.682,Z 142.608,A -85,B 0,C 180,E1 -6512.149,E2 -6512.149} C_VEL
LIN {X 0,Y 488.699,Z 142.613,A -85,B 0,C 180,E1 -6515.117,E2 -6515.117} C_VEL
LIN {X 0,Y 488.648,Z 142.612,A -85,B 0,C 180,E1 -6518.203,E2 -6518.203} C_VEL
LIN {X 0,Y 488.687,Z 142.608,A -85,B 0,C 180,E1 -6520.342,E2 -6520.342} C_VEL
LIN {X 0,Y 488.659,Z 142.612,A -85,B 0,C 180,E1 -6523.658,E2 -6523.658} C_VEL
LIN {X 0,Y 488.66,Z 142.612,A -85,B 0,C 180,E1 -6526.344,E2 -6526.344} C_VEL
LIN {X 0,Y 488.699,Z 142.606,A -85,B 0,C 180,E1 -6529.674,E2 -6529.674} C_VEL
LIN {X 0,Y 488.644,Z 142.621,A -85,B 0,C 180,E1 -6532.839,E2 -6532.839} C_VEL
LIN {X 0,Y 488.711,Z 142.604,A -85,B 0,C 180,E1 -6535.887,E2 -6535.887} C_VEL
LIN {X 0,Y 488.655,Z 142.619,A -85,B 0,C 180,E1 -6538.819,E2 -6538.819} C_VEL
LIN {X 0,Y 488.681,Z 142.609,A -85,B 0,C 180,E1 -6541.668,E2 -6541.668} C_VEL
LIN {X 0,Y 488.669,Z 142.618,A -85,B 0,C 180,E1 -6544.746,E2 -6544.746} C_VEL
LIN {X 0,Y 488.694,Z 142.755,A -85,B 0,C 180,E1 -6544.961,E2 -6544.961} C_VEL
LIN {X 0,Y 490.338,Z 151.188,A -85,B 0,C 180,E1 -6546.536,E2 -6546.536} C_VEL
LIN {X 0,Y 490.532,Z 156.426,A -85,B 0,C 180,E1 -6547.465,E2 -6547.465} C_VEL
LIN {X 0,Y 489.962,Z 171.611,A -85,B 0,C 180,E1 -6550.083,E2 -6550.083} C_VEL
LIN {X 0,Y 489.433,Z 188.043,A -85,B 0,C 180,E1 -6552.881,E2 -6552.881} C_VEL
LIN {X 0,Y 489.295,Z 193.187,A -85,B 0,C 180,E1 -6553.75,E2 -6553.75} C_VEL
LIN {X 0,Y 491.586,Z 209.033,A -85,B 0,C 180,E1 -6554.078,E2 -6554.078} C_VEL
LIN {X 0,Y 490.933,Z 301.479,A -85,B 0,C 180,E1 -6555.519,E2 -6555.519} C_VEL
LIN {X 0,Y 490.593,Z 315.31,A -85,B 0,C 180,E1 -6555.906,E2 -6555.906} C_VEL
LIN {X 0,Y 490.263,Z 327.782,A -85,B 0,C 180,E1 -6556.425,E2 -6556.425} C_VEL
LIN {X 0,Y 489.852,Z 339.405,A -85,B 0,C 180,E1 -6557.078,E2 -6557.078} C_VEL
LIN {X 0,Y 489.482,Z 350.549,A -85,B 0,C 180,E1 -6557.879,E2 -6557.879} C_VEL
LIN {X 0,Y 489.13,Z 361.02,A -85,B 0,C 180,E1 -6558.816,E2 -6558.816} C_VEL
LIN {X 0,Y 488.726,Z 370.424,A -85,B 0,C 180,E1 -6559.855,E2 -6559.855} C_VEL
LIN {X 0,Y 488.414,Z 379.52,A -85,B 0,C 180,E1 -6561.102,E2 -6561.102} C_VEL
LIN {X 0,Y 488.204,Z 386.847,A -85,B 0,C 180,E1 -6562.349,E2 -6562.349} C_VEL
LIN {X 0,Y 488.047,Z 392.409,A -85,B 0,C 180,E1 -6563.525,E2 -6563.525} C_VEL
LIN {X 0,Y 488.013,Z 396.597,A -85,B 0,C 180,E1 -6564.63,E2 -6564.63} C_VEL
LIN {X 0,Y 487.926,Z 400.263,A -85,B 0,C 180,E1 -6565.871,E2 -6565.871} C_VEL
LIN {X 0,Y 487.964,Z 402.157,A -85,B 0,C 180,E1 -6566.698,E2 -6566.698} C_VEL
LIN {X 0,Y 487.909,Z 403.575,A -85,B 0,C 180,E1 -6567.524,E2 -6567.524} C_VEL
LIN {X 0,Y 487.891,Z 404.581,A -85,B 0,C 180,E1 -6568.35,E2 -6568.35} C_VEL
LIN {X 0,Y 487.835,Z 405.192,A -85,B 0,C 180,E1 -6569.175,E2 -6569.175} C_VEL
LIN {X 0,Y 487.822,Z 405.407,A -85,B 0,C 180,E1 -6570.001,E2 -6570.001} C_VEL
LIN {X 0,Y 487.836,Z 405.18,A -85,B 0,C 180,E1 -6570.826,E2 -6570.826} C_VEL
LIN {X 0,Y 487.891,Z 404.556,A -85,B 0,C 180,E1 -6571.652,E2 -6571.652} C_VEL
LIN {X 0,Y 487.909,Z 403.536,A -85,B 0,C 180,E1 -6572.477,E2 -6572.477} C_VEL
LIN {X 0,Y 487.964,Z 402.105,A -85,B 0,C 180,E1 -6573.303,E2 -6573.303} C_VEL
LIN {X 0,Y 487.918,Z 399.104,A -85,B 0,C 180,E1 -6574.545,E2 -6574.545} C_VEL
LIN {X 0,Y 488.011,Z 395.045,A -85,B 0,C 180,E1 -6575.786,E2 -6575.786} C_VEL
LIN {X 0,Y 488.18,Z 388.797,A -85,B 0,C 180,E1 -6577.237,E2 -6577.237} C_VEL
LIN {X 0,Y 488.342,Z 381.981,A -85,B 0,C 180,E1 -6578.484,E2 -6578.484} C_VEL
LIN {X 0,Y 488.614,Z 373.516,A -85,B 0,C 180,E1 -6579.731,E2 -6579.731} C_VEL
LIN {X 0,Y 488.97,Z 364.791,A -85,B 0,C 180,E1 -6580.77,E2 -6580.77} C_VEL
LIN {X 0,Y 489.353,Z 354.043,A -85,B 0,C 180,E1 -6581.81,E2 -6581.81} C_VEL
LIN {X 0,Y 489.704,Z 342.393,A -85,B 0,C 180,E1 -6582.711,E2 -6582.711} C_VEL
LIN {X 0,Y 490.179,Z 329.505,A -85,B 0,C 180,E1 -6583.474,E2 -6583.474} C_VEL
LIN {X 0,Y 490.572,Z 316.547,A -85,B 0,C 180,E1 -6584.044,E2 -6584.044} C_VEL
LIN {X 0,Y 490.909,Z 303.506,A -85,B 0,C 180,E1 -6584.43,E2 -6584.43} C_VEL
LIN {X 0,Y 491.127,Z 282.14,A -85,B 0,C 180,E1 -6584.795,E2 -6584.795} C_VEL
LIN {X 0,Y 491.576,Z 207.941,A -85,B 0,C 180,E1 -6585.957,E2 -6585.957} C_VEL
LIN {X 0,Y 489.223,Z 192.472,A -85,B 0,C 180,E1 -6586.301,E2 -6586.301} C_VEL
LIN {X 0,Y 489.745,Z 174.62,A -85,B 0,C 180,E1 -6589.273,E2 -6589.273} C_VEL
LIN {X 0,Y 490.269,Z 157.842,A -85,B 0,C 180,E1 -6592.105,E2 -6592.105} C_VEL
LIN {X 0,Y 490.387,Z 152.115,A -85,B 0,C 180,E1 -6593.081,E2 -6593.081} C_VEL
LIN {X 0,Y 488.688,Z 142.615,A -85,B 0,C 180,E1 -6594.844,E2 -6594.844} C_VEL
LIN {X 0,Y 488.677,Z 142.618,A -85,B 0,C 180,E1 -6597.402,E2 -6597.402} C_VEL
LIN {X 0,Y 488.654,Z 142.614,A -85,B 0,C 180,E1 -6600.351,E2 -6600.351} C_VEL
LIN {X 0,Y 488.71,Z 142.61,A -85,B 0,C 180,E1 -6603.48,E2 -6603.48} C_VEL
LIN {X 0,Y 488.654,Z 142.614,A -85,B 0,C 180,E1 -6606.35,E2 -6606.35} C_VEL
LIN {X 0,Y 488.689,Z 142.613,A -85,B 0,C 180,E1 -6609.256,E2 -6609.256} C_VEL
LIN {X 0,Y 488.669,Z 142.611,A -85,B 0,C 180,E1 -6611.595,E2 -6611.595} C_VEL
LIN {X 0,Y 488.704,Z 142.611,A -85,B 0,C 180,E1 -6614.803,E2 -6614.803} C_VEL
LIN {X 0,Y 488.652,Z 142.611,A -85,B 0,C 180,E1 -6617.47,E2 -6617.47} C_VEL
LIN {X 0,Y 488.707,Z 142.604,A -85,B 0,C 180,E1 -6619.674,E2 -6619.674} C_VEL
LIN {X 0,Y 488.668,Z 142.615,A -85,B 0,C 180,E1 -6622.84,E2 -6622.84} C_VEL
LIN {X 0,Y 488.72,Z 142.605,A -85,B 0,C 180,E1 -6625.886,E2 -6625.886} C_VEL
LIN {X 0,Y 488.685,Z 142.61,A -85,B 0,C 180,E1 -6628.82,E2 -6628.82} C_VEL
LIN {X 0,Y 488.694,Z 142.607,A -85,B 0,C 180,E1 -6631.668,E2 -6631.668} C_VEL
LIN {X 0,Y 488.693,Z 142.612,A -85,B 0,C 180,E1 -6634.441,E2 -6634.441} C_VEL
LIN {X 0,Y 488.724,Z 142.602,A -85,B 0,C 180,E1 -6637.153,E2 -6637.153} C_VEL
LIN {X 0,Y 488.722,Z 142.605,A -85,B 0,C 180,E1 -6639.81,E2 -6639.81} C_VEL
LIN {X 0,Y 488.681,Z 142.614,A -85,B 0,C 180,E1 -6642.422,E2 -6642.422} C_VEL
LIN {X 0,Y 488.754,Z 142.601,A -85,B 0,C 180,E1 -6644.999,E2 -6644.999} C_VEL
LIN {X 0,Y 488.809,Z 142.598,A -85,B 0,C 180,E1 -6648.388,E2 -6648.388} C_VEL
LIN {X 0,Y 488.765,Z 142.606,A -85,B 0,C 180,E1 -6651.733,E2 -6651.733} C_VEL
LIN {X 0,Y 488.818,Z 142.596,A -85,B 0,C 180,E1 -6654.224,E2 -6654.224} C_VEL
LIN {X 0,Y 488.947,Z 142.583,A -85,B 0,C 180,E1 -6657.529,E2 -6657.529} C_VEL
LIN {X 0,Y 488.948,Z 142.583,A -85,B 0,C 180,E1 -6660,E2 -6660} C_VEL
LIN {X 0,Y 488.956,Z 142.579,A -85,B 0,C 180,E1 -6662.472,E2 -6662.472} C_VEL
LIN {X 0,Y 488.834,Z 142.598,A -85,B 0,C 180,E1 -6665.776,E2 -6665.776} C_VEL
LIN {X 0,Y 488.851,Z 142.767,A -85,B 0,C 180,E1 -6667.071,E2 -6667.071} C_VEL
LIN {X 0,Y 489.697,Z 148.918,A -85,B 0,C 180,E1 -6668.252,E2 -6668.252} C_VEL
LIN {X 0,Y 489.478,Z 163.651,A -85,B 0,C 180,E1 -6670.967,E2 -6670.967} C_VEL
LIN {X 0,Y 489.429,Z 168.01,A -85,B 0,C 180,E1 -6671.772,E2 -6671.772} C_VEL
LIN {X 0,Y 491.842,Z 181.688,A -85,B 0,C 180,E1 -6672.084,E2 -6672.084} C_VEL
LIN {X 0,Y 490.974,Z 276.292,A -85,B 0,C 180,E1 -6673.582,E2 -6673.582} C_VEL
LIN {X 0,Y 490.71,Z 289.449,A -85,B 0,C 180,E1 -6673.96,E2 -6673.96} C_VEL
LIN {X 0,Y 490.443,Z 301.598,A -85,B 0,C 180,E1 -6674.471,E2 -6674.471} C_VEL
LIN {X 0,Y 490.074,Z 313.895,A -85,B 0,C 180,E1 -6675.172,E2 -6675.172} C_VEL
LIN {X 0,Y 489.648,Z 325.435,A -85,B 0,C 180,E1 -6676.02,E2 -6676.02} C_VEL
LIN {X 0,Y 489.237,Z 336.221,A -85,B 0,C 180,E1 -6677.019,E2 -6677.019} C_VEL
LIN {X 0,Y 488.867,Z 345.942,A -85,B 0,C 180,E1 -6678.144,E2 -6678.144} C_VEL
LIN {X 0,Y 488.576,Z 354.187,A -85,B 0,C 180,E1 -6679.321,E2 -6679.321} C_VEL
LIN {X 0,Y 488.288,Z 361.765,A -85,B 0,C 180,E1 -6680.681,E2 -6680.681} C_VEL
LIN {X 0,Y 488.129,Z 367.48,A -85,B 0,C 180,E1 -6681.984,E2 -6681.984} C_VEL
LIN {X 0,Y 488.012,Z 372.029,A -85,B 0,C 180,E1 -6683.331,E2 -6683.331} C_VEL
LIN {X 0,Y 487.87,Z 375.64,A -85,B 0,C 180,E1 -6684.831,E2 -6684.831} C_VEL
LIN {X 0,Y 487.831,Z 376.925,A -85,B 0,C 180,E1 -6685.608,E2 -6685.608} C_VEL
LIN {X 0,Y 487.805,Z 378.166,A -85,B 0,C 180,E1 -6686.713,E2 -6686.713} C_VEL
LIN {X 0,Y 487.788,Z 378.572,A -85,B 0,C 180,E1 -6687.455,E2 -6687.455} C_VEL
LIN {X 0,Y 487.83,Z 378.584,A -85,B 0,C 180,E1 -6688.5,E2 -6688.5} C_VEL
LIN {X 0,Y 487.833,Z 378.168,A -85,B 0,C 180,E1 -6689.329,E2 -6689.329} C_VEL
LIN {X 0,Y 487.884,Z 377.148,A -85,B 0,C 180,E1 -6690.277,E2 -6690.277} C_VEL
LIN {X 0,Y 487.956,Z 374.382,A -85,B 0,C 180,E1 -6691.812,E2 -6691.812} C_VEL
LIN {X 0,Y 488.007,Z 370.653,A -85,B 0,C 180,E1 -6693.179,E2 -6693.179} C_VEL
LIN {X 0,Y 488.159,Z 365.747,A -85,B 0,C 180,E1 -6694.506,E2 -6694.506} C_VEL
LIN {X 0,Y 488.382,Z 359.031,A -85,B 0,C 180,E1 -6695.903,E2 -6695.903} C_VEL
LIN {X 0,Y 488.679,Z 351.424,A -85,B 0,C 180,E1 -6697.159,E2 -6697.159} C_VEL
LIN {X 0,Y 488.97,Z 342.833,A -85,B 0,C 180,E1 -6698.305,E2 -6698.305} C_VEL
LIN {X 0,Y 489.332,Z 333.379,A -85,B 0,C 180,E1 -6699.327,E2 -6699.327} C_VEL
LIN {X 0,Y 489.685,Z 321.947,A -85,B 0,C 180,E1 -6700.327,E2 -6700.327} C_VEL
LIN {X 0,Y 490.106,Z 311.518,A -85,B 0,C 180,E1 -6701.048,E2 -6701.048} C_VEL
LIN {X 0,Y 490.418,Z 302.691,A -85,B 0,C 180,E1 -6701.541,E2 -6701.541} C_VEL
LIN {X 0,Y 489.955,Z 297.303,A -85,B 0,C 180,E1 -6701.822,E2 -6701.822} C_VEL
LIN {X 0,Y 487.306,Z 288.469,A -85,B 0,C 180,E1 -6702.257,E2 -6702.257} C_VEL
LIN {X 0,Y 484.62,Z 279.403,A -85,B 0,C 180,E1 -6702.605,E2 -6702.605} C_VEL
LIN {X 0,Y 484.089,Z 273.656,A -85,B 0,C 180,E1 -6702.746,E2 -6702.746} C_VEL
LIN {X 0,Y 484.829,Z 181.292,A -85,B 0,C 180,E1 -6704.206,E2 -6704.206} C_VEL
LIN {X 0,Y 482.35,Z 168.022,A -85,B 0,C 180,E1 -6704.515,E2 -6704.515} C_VEL
LIN {X 0,Y 482.896,Z 152.214,A -85,B 0,C 180,E1 -6707.692,E2 -6707.692} C_VEL
LIN {X 0,Y 482.374,Z 147.153,A -85,B 0,C 180,E1 -6708.755,E2 -6708.755} C_VEL
LIN {X 0,Y 481.699,Z 143.483,A -85,B 0,C 180,E1 -6709.552,E2 -6709.552} C_VEL
LIN {X 0,Y 481.618,Z 143.493,A -85,B 0,C 180,E1 -6712.201,E2 -6712.201} C_VEL
LIN {X 0,Y 481.686,Z 143.48,A -85,B 0,C 180,E1 -6715.317,E2 -6715.317} C_VEL
LIN {X 0,Y 481.641,Z 143.491,A -85,B 0,C 180,E1 -6718.311,E2 -6718.311} C_VEL
LIN {X 0,Y 481.643,Z 143.485,A -85,B 0,C 180,E1 -6721.214,E2 -6721.214} C_VEL
LIN {X 0,Y 481.631,Z 143.49,A -85,B 0,C 180,E1 -6724.038,E2 -6724.038} C_VEL
LIN {X 0,Y 481.657,Z 143.485,A -85,B 0,C 180,E1 -6726.818,E2 -6726.818} C_VEL
LIN {X 0,Y 481.662,Z 143.483,A -85,B 0,C 180,E1 -6729.501,E2 -6729.501} C_VEL
LIN {X 0,Y 481.655,Z 143.492,A -85,B 0,C 180,E1 -6732.156,E2 -6732.156} C_VEL
LIN {X 0,Y 481.727,Z 143.475,A -85,B 0,C 180,E1 -6734.775,E2 -6734.775} C_VEL
LIN {X 0,Y 481.741,Z 143.479,A -85,B 0,C 180,E1 -6738.214,E2 -6738.214} C_VEL
LIN {X 0,Y 481.721,Z 143.478,A -85,B 0,C 180,E1 -6741.61,E2 -6741.61} C_VEL
LIN {X 0,Y 481.777,Z 143.474,A -85,B 0,C 180,E1 -6744.138,E2 -6744.138} C_VEL
LIN {X 0,Y 481.911,Z 143.455,A -85,B 0,C 180,E1 -6747.492,E2 -6747.492} C_VEL
LIN {X 0,Y 481.914,Z 143.457,A -85,B 0,C 180,E1 -6749.999,E2 -6749.999} C_VEL
LIN {X 0,Y 481.91,Z 143.452,A -85,B 0,C 180,E1 -6752.507,E2 -6752.507} C_VEL
LIN {X 0,Y 481.769,Z 143.475,A -85,B 0,C 180,E1 -6755.86,E2 -6755.86} C_VEL
LIN {X 0,Y 481.719,Z 143.476,A -85,B 0,C 180,E1 -6758.388,E2 -6758.388} C_VEL
LIN {X 0,Y 481.738,Z 143.478,A -85,B 0,C 180,E1 -6761.784,E2 -6761.784} C_VEL
LIN {X 0,Y 481.73,Z 143.478,A -85,B 0,C 180,E1 -6765.224,E2 -6765.224} C_VEL
LIN {X 0,Y 481.651,Z 143.484,A -85,B 0,C 180,E1 -6768.723,E2 -6768.723} C_VEL
LIN {X 0,Y 481.631,Z 143.494,A -85,B 0,C 180,E1 -6771.395,E2 -6771.395} C_VEL
LIN {X 0,Y 481.646,Z 143.485,A -85,B 0,C 180,E1 -6774.114,E2 -6774.114} C_VEL
LIN {X 0,Y 481.651,Z 143.49,A -85,B 0,C 180,E1 -6777.116,E2 -6777.116} C_VEL
LIN {X 0,Y 481.65,Z 143.486,A -85,B 0,C 180,E1 -6779.742,E2 -6779.742} C_VEL
LIN {X 0,Y 481.648,Z 143.487,A -85,B 0,C 180,E1 -6782.675,E2 -6782.675} C_VEL
LIN {X 0,Y 481.626,Z 143.488,A -85,B 0,C 180,E1 -6785.709,E2 -6785.709} C_VEL
LIN {X 0,Y 481.663,Z 143.489,A -85,B 0,C 180,E1 -6788.859,E2 -6788.859} C_VEL
LIN {X 0,Y 481.612,Z 143.489,A -85,B 0,C 180,E1 -6792.163,E2 -6792.163} C_VEL
LIN {X 0,Y 481.65,Z 143.487,A -85,B 0,C 180,E1 -6794.457,E2 -6794.457} C_VEL
LIN {X 0,Y 481.612,Z 143.497,A -85,B 0,C 180,E1 -6796.854,E2 -6796.854} C_VEL
LIN {X 0,Y 481.651,Z 143.484,A -85,B 0,C 180,E1 -6800.056,E2 -6800.056} C_VEL
LIN {X 0,Y 481.613,Z 143.49,A -85,B 0,C 180,E1 -6803.251,E2 -6803.251} C_VEL
LIN {X 0,Y 481.665,Z 143.486,A -85,B 0,C 180,E1 -6806.326,E2 -6806.326} C_VEL
LIN {X 0,Y 481.628,Z 143.487,A -85,B 0,C 180,E1 -6809.42,E2 -6809.42} C_VEL
LIN {X 0,Y 481.641,Z 143.489,A -85,B 0,C 180,E1 -6812.164,E2 -6812.164} C_VEL
LIN {X 0,Y 481.666,Z 143.484,A -85,B 0,C 180,E1 -6814.967,E2 -6814.967} C_VEL
LIN {X 0,Y 481.629,Z 143.487,A -85,B 0,C 180,E1 -6817.703,E2 -6817.703} C_VEL
LIN {X 0,Y 481.686,Z 143.487,A -85,B 0,C 180,E1 -6820.392,E2 -6820.392} C_VEL
LIN {X 0,Y 481.608,Z 143.49,A -85,B 0,C 180,E1 -6823.031,E2 -6823.031} C_VEL
LIN {X 0,Y 481.664,Z 143.483,A -85,B 0,C 180,E1 -6825.638,E2 -6825.638} C_VEL
LIN {X 0,Y 481.728,Z 143.482,A -85,B 0,C 180,E1 -6828.214,E2 -6828.214} C_VEL
LIN {X 0,Y 481.708,Z 143.479,A -85,B 0,C 180,E1 -6831.61,E2 -6831.61} C_VEL
LIN {X 0,Y 481.768,Z 143.477,A -85,B 0,C 180,E1 -6834.139,E2 -6834.139} C_VEL
LIN {X 0,Y 481.899,Z 143.455,A -85,B 0,C 180,E1 -6837.492,E2 -6837.492} C_VEL
LIN {X 0,Y 481.902,Z 143.46,A -85,B 0,C 180,E1 -6840,E2 -6840} C_VEL
LIN {X 0,Y 481.898,Z 143.454,A -85,B 0,C 180,E1 -6842.507,E2 -6842.507} C_VEL
LIN {X 0,Y 481.764,Z 143.478,A -85,B 0,C 180,E1 -6845.861,E2 -6845.861} C_VEL
LIN {X 0,Y 481.707,Z 143.478,A -85,B 0,C 180,E1 -6848.389,E2 -6848.389} C_VEL
LIN {X 0,Y 481.727,Z 143.482,A -85,B 0,C 180,E1 -6851.785,E2 -6851.785} C_VEL
LIN {X 0,Y 481.72,Z 143.478,A -85,B 0,C 180,E1 -6855.225,E2 -6855.225} C_VEL
LIN {X 0,Y 481.641,Z 143.485,A -85,B 0,C 180,E1 -6858.724,E2 -6858.724} C_VEL
LIN {X 0,Y 481.621,Z 143.494,A -85,B 0,C 180,E1 -6861.396,E2 -6861.396} C_VEL
LIN {X 0,Y 481.633,Z 143.487,A -85,B 0,C 180,E1 -6864.115,E2 -6864.115} C_VEL
LIN {X 0,Y 481.643,Z 143.49,A -85,B 0,C 180,E1 -6867.117,E2 -6867.117} C_VEL
LIN {X 0,Y 481.592,Z 143.494,A -85,B 0,C 180,E1 -6869.747,E2 -6869.747} C_VEL
LIN {X 0,Y 481.642,Z 143.486,A -85,B 0,C 180,E1 -6872.676,E2 -6872.676} C_VEL
LIN {X 0,Y 481.643,Z 143.493,A -85,B 0,C 180,E1 -6875.202,E2 -6875.202} C_VEL
LIN {X 0,Y 481.623,Z 143.487,A -85,B 0,C 180,E1 -6878.004,E2 -6878.004} C_VEL
LIN {X 0,Y 481.616,Z 143.496,A -85,B 0,C 180,E1 -6881.046,E2 -6881.046} C_VEL
LIN {X 0,Y 481.644,Z 143.486,A -85,B 0,C 180,E1 -6884.459,E2 -6884.459} C_VEL
LIN {X 0,Y 481.606,Z 143.496,A -85,B 0,C 180,E1 -6886.856,E2 -6886.856} C_VEL
LIN {X 0,Y 481.65,Z 143.484,A -85,B 0,C 180,E1 -6890.058,E2 -6890.058} C_VEL
LIN {X 0,Y 481.602,Z 143.492,A -85,B 0,C 180,E1 -6893.38,E2 -6893.38} C_VEL
LIN {X 0,Y 481.667,Z 143.484,A -85,B 0,C 180,E1 -6896.328,E2 -6896.328} C_VEL
LIN {X 0,Y 481.607,Z 143.491,A -85,B 0,C 180,E1 -6899.427,E2 -6899.427} C_VEL
LIN {X 0,Y 481.64,Z 143.489,A -85,B 0,C 180,E1 -6902.165,E2 -6902.165} C_VEL
LIN {X 0,Y 481.658,Z 143.669,A -85,B 0,C 180,E1 -6904.778,E2 -6904.778} C_VEL
LIN {X 0,Y 483.528,Z 153.483,A -85,B 0,C 180,E1 -6906.636,E2 -6906.636} C_VEL
LIN {X 0,Y 483.425,Z 161.214,A -85,B 0,C 180,E1 -6908.007,E2 -6908.007} C_VEL
LIN {X 0,Y 482.868,Z 177.563,A -85,B 0,C 180,E1 -6910.858,E2 -6910.858} C_VEL
LIN {X 0,Y 482.297,Z 193.127,A -85,B 0,C 180,E1 -6913.522,E2 -6913.522} C_VEL
LIN {X 0,Y 484.726,Z 209.563,A -85,B 0,C 180,E1 -6913.868,E2 -6913.868} C_VEL
LIN {X 0,Y 484.039,Z 301.74,A -85,B 0,C 180,E1 -6915.335,E2 -6915.335} C_VEL
LIN {X 0,Y 483.684,Z 315.409,A -85,B 0,C 180,E1 -6915.727,E2 -6915.727} C_VEL
LIN {X 0,Y 483.324,Z 327.246,A -85,B 0,C 180,E1 -6916.226,E2 -6916.226} C_VEL
LIN {X 0,Y 482.942,Z 338.496,A -85,B 0,C 180,E1 -6916.858,E2 -6916.858} C_VEL
LIN {X 0,Y 482.496,Z 349.767,A -85,B 0,C 180,E1 -6917.669,E2 -6917.669} C_VEL
LIN {X 0,Y 482.078,Z 360.664,A -85,B 0,C 180,E1 -6918.65,E2 -6918.65} C_VEL
LIN {X 0,Y 481.7,Z 370.118,A -85,B 0,C 180,E1 -6919.705,E2 -6919.705} C_VEL
LIN {X 0,Y 481.367,Z 379.242,A -85,B 0,C 180,E1 -6920.971,E2 -6920.971} C_VEL
LIN {X 0,Y 481.132,Z 386.591,A -85,B 0,C 180,E1 -6922.235,E2 -6922.235} C_VEL
LIN {X 0,Y 480.943,Z 392.708,A -85,B 0,C 180,E1 -6923.557,E2 -6923.557} C_VEL
LIN {X 0,Y 480.894,Z 397.719,A -85,B 0,C 180,E1 -6924.97,E2 -6924.97} C_VEL
LIN {X 0,Y 480.826,Z 400.051,A -85,B 0,C 180,E1 -6925.81,E2 -6925.81} C_VEL
LIN {X 0,Y 480.887,Z 401.951,A -85,B 0,C 180,E1 -6926.649,E2 -6926.649} C_VEL
LIN {X 0,Y 480.823,Z 403.374,A -85,B 0,C 180,E1 -6927.488,E2 -6927.488} C_VEL
LIN {X 0,Y 480.792,Z 404.383,A -85,B 0,C 180,E1 -6928.325,E2 -6928.325} C_VEL
LIN {X 0,Y 480.761,Z 404.996,A -85,B 0,C 180,E1 -6929.163,E2 -6929.163} C_VEL
LIN {X 0,Y 480.746,Z 405.213,A -85,B 0,C 180,E1 -6930.001,E2 -6930.001} C_VEL
LIN {X 0,Y 480.761,Z 404.987,A -85,B 0,C 180,E1 -6930.838,E2 -6930.838} C_VEL
LIN {X 0,Y 480.792,Z 404.361,A -85,B 0,C 180,E1 -6931.676,E2 -6931.676} C_VEL
LIN {X 0,Y 480.823,Z 403.34,A -85,B 0,C 180,E1 -6932.514,E2 -6932.514} C_VEL
LIN {X 0,Y 480.888,Z 401.908,A -85,B 0,C 180,E1 -6933.352,E2 -6933.352} C_VEL
LIN {X 0,Y 480.837,Z 398.902,A -85,B 0,C 180,E1 -6934.612,E2 -6934.612} C_VEL
LIN {X 0,Y 480.916,Z 394.839,A -85,B 0,C 180,E1 -6935.872,E2 -6935.872} C_VEL
LIN {X 0,Y 481.104,Z 388.582,A -85,B 0,C 180,E1 -6937.344,E2 -6937.344} C_VEL
LIN {X 0,Y 481.297,Z 381.753,A -85,B 0,C 180,E1 -6938.609,E2 -6938.609} C_VEL
LIN {X 0,Y 481.55,Z 373.277,A -85,B 0,C 180,E1 -6939.875,E2 -6939.875} C_VEL
LIN {X 0,Y 481.97,Z 364.547,A -85,B 0,C 180,E1 -6940.928,E2 -6940.928} C_VEL
LIN {X 0,Y 482.376,Z 354.011,A -85,B 0,C 180,E1 -6941.964,E2 -6941.964} C_VEL
LIN {X 0,Y 482.708,Z 343.415,A -85,B 0,C 180,E1 -6942.808,E2 -6942.808} C_VEL
LIN {X 0,Y 483.2,Z 331.246,A -85,B 0,C 180,E1 -6943.565,E2 -6943.565} C_VEL
LIN {X 0,Y 483.593,Z 318.934,A -85,B 0,C 180,E1 -6944.143,E2 -6944.143} C_VEL
LIN {X 0,Y 483.921,Z 306.423,A -85,B 0,C 180,E1 -6944.563,E2 -6944.563} C_VEL
LIN {X 0,Y 484.198,Z 292.126,A -85,B 0,C 180,E1 -6944.85,E2 -6944.85} C_VEL
LIN {X 0,Y 484.788,Z 208.63,A -85,B 0,C 180,E1 -6946.182,E2 -6946.182} C_VEL
LIN {X 0,Y 482.223,Z 192.188,A -85,B 0,C 180,E1 -6946.566,E2 -6946.566} C_VEL
LIN {X 0,Y 482.763,Z 175.743,A -85,B 0,C 180,E1 -6949.349,E2 -6949.349} C_VEL
LIN {X 0,Y 483.325,Z 158.99,A -85,B 0,C 180,E1 -6952.214,E2 -6952.214} C_VEL
LIN {X 0,Y 483.458,Z 153.804,A -85,B 0,C 180,E1 -6953.111,E2 -6953.111} C_VEL
LIN {X 0,Y 481.755,Z 144.096,A -85,B 0,C 180,E1 -6954.913,E2 -6954.913} C_VEL
LIN {X 0,Y 481.667,Z 143.49,A -85,B 0,C 180,E1 -6955.034,E2 -6955.034} C_VEL
LIN {X 0,Y 481.644,Z 143.491,A -85,B 0,C 180,E1 -6957.836,E2 -6957.836} C_VEL
LIN {X 0,Y 481.611,Z 143.493,A -85,B 0,C 180,E1 -6960.714,E2 -6960.714} C_VEL
LIN {X 0,Y 481.678,Z 143.484,A -85,B 0,C 180,E1 -6963.729,E2 -6963.729} C_VEL
LIN {X 0,Y 481.61,Z 143.495,A -85,B 0,C 180,E1 -6966.749,E2 -6966.749} C_VEL
LIN {X 0,Y 481.658,Z 143.484,A -85,B 0,C 180,E1 -6969.943,E2 -6969.943} C_VEL
LIN {X 0,Y 481.621,Z 143.49,A -85,B 0,C 180,E1 -6973.303,E2 -6973.303} C_VEL
LIN {X 0,Y 481.655,Z 143.482,A -85,B 0,C 180,E1 -6975.642,E2 -6975.642} C_VEL
LIN {X 0,Y 481.625,Z 143.49,A -85,B 0,C 180,E1 -6978.955,E2 -6978.955} C_VEL
LIN {X 0,Y 481.641,Z 143.485,A -85,B 0,C 180,E1 -6981.996,E2 -6981.996} C_VEL
LIN {X 0,Y 481.683,Z 143.482,A -85,B 0,C 180,E1 -6985.317,E2 -6985.317} C_VEL
LIN {X 0,Y 481.641,Z 143.492,A -85,B 0,C 180,E1 -6988.311,E2 -6988.311} C_VEL
LIN {X 0,Y 481.655,Z 143.483,A -85,B 0,C 180,E1 -6991.216,E2 -6991.216} C_VEL
LIN {X 0,Y 481.645,Z 143.489,A -85,B 0,C 180,E1 -6994.04,E2 -6994.04} C_VEL
LIN {X 0,Y 481.657,Z 143.484,A -85,B 0,C 180,E1 -6996.818,E2 -6996.818} C_VEL
LIN {X 0,Y 481.696,Z 143.478,A -85,B 0,C 180,E1 -6999.503,E2 -6999.503} C_VEL
LIN {X 0,Y 481.672,Z 143.488,A -85,B 0,C 180,E1 -7002.157,E2 -7002.157} C_VEL
LIN {X 0,Y 481.734,Z 143.476,A -85,B 0,C 180,E1 -7004.776,E2 -7004.776} C_VEL
LIN {X 0,Y 481.755,Z 143.478,A -85,B 0,C 180,E1 -7008.215,E2 -7008.215} C_VEL
LIN {X 0,Y 481.724,Z 143.483,A -85,B 0,C 180,E1 -7011.611,E2 -7011.611} C_VEL
LIN {X 0,Y 481.779,Z 143.474,A -85,B 0,C 180,E1 -7014.139,E2 -7014.139} C_VEL
LIN {X 0,Y 481.912,Z 143.459,A -85,B 0,C 180,E1 -7017.493,E2 -7017.493} C_VEL
LIN {X 0,Y 481.917,Z 143.459,A -85,B 0,C 180,E1 -7020,E2 -7020} C_VEL
LIN {X 0,Y 481.922,Z 143.455,A -85,B 0,C 180,E1 -7022.508,E2 -7022.508} C_VEL
LIN {X 0,Y 481.794,Z 143.474,A -85,B 0,C 180,E1 -7025.861,E2 -7025.861} C_VEL
LIN {X 0,Y 481.791,Z 143.618,A -85,B 0,C 180,E1 -7026.877,E2 -7026.877} C_VEL
LIN {X 0,Y 482.77,Z 150.1,A -85,B 0,C 180,E1 -7028.138,E2 -7028.138} C_VEL
LIN {X 0,Y 482.511,Z 164.993,A -85,B 0,C 180,E1 -7030.915,E2 -7030.915} C_VEL
LIN {X 0,Y 482.462,Z 168.129,A -85,B 0,C 180,E1 -7031.501,E2 -7031.501} C_VEL
LIN {X 0,Y 484.994,Z 181.7,A -85,B 0,C 180,E1 -7031.838,E2 -7031.838} C_VEL
LIN {X 0,Y 484.119,Z 276.603,A -85,B 0,C 180,E1 -7033.376,E2 -7033.376} C_VEL
LIN {X 0,Y 483.836,Z 289.747,A -85,B 0,C 180,E1 -7033.76,E2 -7033.76} C_VEL
LIN {X 0,Y 483.529,Z 302.407,A -85,B 0,C 180,E1 -7034.306,E2 -7034.306} C_VEL
LIN {X 0,Y 483.191,Z 313.72,A -85,B 0,C 180,E1 -7034.962,E2 -7034.962} C_VEL
LIN {X 0,Y 482.712,Z 325.599,A -85,B 0,C 180,E1 -7035.842,E2 -7035.842} C_VEL
LIN {X 0,Y 482.281,Z 336.203,A -85,B 0,C 180,E1 -7036.836,E2 -7036.836} C_VEL
LIN {X 0,Y 481.851,Z 346.271,A -85,B 0,C 180,E1 -7038.017,E2 -7038.017} C_VEL
LIN {X 0,Y 481.548,Z 354.239,A -85,B 0,C 180,E1 -7039.171,E2 -7039.171} C_VEL
LIN {X 0,Y 481.295,Z 360.578,A -85,B 0,C 180,E1 -7040.292,E2 -7040.292} C_VEL
LIN {X 0,Y 481.13,Z 365.789,A -85,B 0,C 180,E1 -7041.419,E2 -7041.419} C_VEL
LIN {X 0,Y 480.967,Z 370.375,A -85,B 0,C 180,E1 -7042.653,E2 -7042.653} C_VEL
LIN {X 0,Y 480.867,Z 374.534,A -85,B 0,C 180,E1 -7044.157,E2 -7044.157} C_VEL
LIN {X 0,Y 480.756,Z 376.363,A -85,B 0,C 180,E1 -7045.084,E2 -7045.084} C_VEL
LIN {X 0,Y 480.719,Z 377.717,A -85,B 0,C 180,E1 -7046.015,E2 -7046.015} C_VEL
LIN {X 0,Y 480.705,Z 378.519,A -85,B 0,C 180,E1 -7046.951,E2 -7046.951} C_VEL
LIN {X 0,Y 480.701,Z 378.849,A -85,B 0,C 180,E1 -7047.895,E2 -7047.895} C_VEL
LIN {X 0,Y 480.727,Z 378.657,A -85,B 0,C 180,E1 -7048.846,E2 -7048.846} C_VEL
LIN {X 0,Y 480.811,Z 377.191,A -85,B 0,C 180,E1 -7050.412,E2 -7050.412} C_VEL
LIN {X 0,Y 480.886,Z 374.164,A -85,B 0,C 180,E1 -7052.042,E2 -7052.042} C_VEL
LIN {X 0,Y 480.989,Z 369.627,A -85,B 0,C 180,E1 -7053.606,E2 -7053.606} C_VEL
LIN {X 0,Y 481.098,Z 365.319,A -85,B 0,C 180,E1 -7054.731,E2 -7054.731} C_VEL
LIN {X 0,Y 481.361,Z 358.358,A -85,B 0,C 180,E1 -7056.165,E2 -7056.165} C_VEL
LIN {X 0,Y 481.647,Z 351.668,A -85,B 0,C 180,E1 -7057.269,E2 -7057.269} C_VEL
LIN {X 0,Y 481.933,Z 343.421,A -85,B 0,C 180,E1 -7058.392,E2 -7058.392} C_VEL
LIN {X 0,Y 482.33,Z 333.912,A -85,B 0,C 180,E1 -7059.442,E2 -7059.442} C_VEL
LIN {X 0,Y 482.666,Z 323.377,A -85,B 0,C 180,E1 -7060.388,E2 -7060.388} C_VEL
LIN {X 0,Y 483.155,Z 311.509,A -85,B 0,C 180,E1 -7061.233,E2 -7061.233} C_VEL
LIN {X 0,Y 483.555,Z 299.498,A -85,B 0,C 180,E1 -7061.887,E2 -7061.887} C_VEL
LIN {X 0,Y 483.851,Z 286.729,A -85,B 0,C 180,E1 -7062.401,E2 -7062.401} C_VEL
LIN {X 0,Y 484.089,Z 273.656,A -85,B 0,C 180,E1 -7062.746,E2 -7062.746} C_VEL
LIN {X 0,Y 483.573,Z 267.865,A -85,B 0,C 180,E1 -7062.866,E2 -7062.866} C_VEL
LIN {X 0,Y 478.111,Z 249.181,A -85,B 0,C 180,E1 -7063.324,E2 -7063.324} C_VEL
LIN {X 0,Y 477.467,Z 243.374,A -85,B 0,C 180,E1 -7063.435,E2 -7063.435} C_VEL
LIN {X 0,Y 478.044,Z 182.431,A -85,B 0,C 180,E1 -7064.412,E2 -7064.412} C_VEL
LIN {X 0,Y 475.398,Z 168.134,A -85,B 0,C 180,E1 -7064.759,E2 -7064.759} C_VEL
LIN {X 0,Y 475.91,Z 154.206,A -85,B 0,C 180,E1 -7067.594,E2 -7067.594} C_VEL
LIN {X 0,Y 475.497,Z 148.96,A -85,B 0,C 180,E1 -7068.703,E2 -7068.703} C_VEL
LIN {X 0,Y 474.652,Z 144.361,A -85,B 0,C 180,E1 -7069.754,E2 -7069.754} C_VEL
LIN {X 0,Y 474.568,Z 144.37,A -85,B 0,C 180,E1 -7073.102,E2 -7073.102} C_VEL
LIN {X 0,Y 474.626,Z 144.361,A -85,B 0,C 180,E1 -7076.019,E2 -7076.019} C_VEL
LIN {X 0,Y 474.59,Z 144.367,A -85,B 0,C 180,E1 -7078.781,E2 -7078.781} C_VEL
LIN {X 0,Y 474.598,Z 144.363,A -85,B 0,C 180,E1 -7081.714,E2 -7081.714} C_VEL
LIN {X 0,Y 474.604,Z 144.366,A -85,B 0,C 180,E1 -7084.596,E2 -7084.596} C_VEL
LIN {X 0,Y 474.588,Z 144.364,A -85,B 0,C 180,E1 -7087.354,E2 -7087.354} C_VEL
LIN {X 0,Y 474.617,Z 144.366,A -85,B 0,C 180,E1 -7090.087,E2 -7090.087} C_VEL
LIN {X 0,Y 474.59,Z 144.365,A -85,B 0,C 180,E1 -7092.772,E2 -7092.772} C_VEL
LIN {X 0,Y 474.631,Z 144.359,A -85,B 0,C 180,E1 -7095.42,E2 -7095.42} C_VEL
LIN {X 0,Y 474.699,Z 144.358,A -85,B 0,C 180,E1 -7098.037,E2 -7098.037} C_VEL
LIN {X 0,Y 474.67,Z 144.356,A -85,B 0,C 180,E1 -7101.485,E2 -7101.485} C_VEL
LIN {X 0,Y 474.74,Z 144.351,A -85,B 0,C 180,E1 -7104.051,E2 -7104.051} C_VEL
LIN {X 0,Y 474.875,Z 144.331,A -85,B 0,C 180,E1 -7107.455,E2 -7107.455} C_VEL
LIN {X 0,Y 474.884,Z 144.332,A -85,B 0,C 180,E1 -7109.999,E2 -7109.999} C_VEL
LIN {X 0,Y 474.875,Z 144.328,A -85,B 0,C 180,E1 -7112.544,E2 -7112.544} C_VEL
LIN {X 0,Y 474.732,Z 144.35,A -85,B 0,C 180,E1 -7115.947,E2 -7115.947} C_VEL
LIN {X 0,Y 474.668,Z 144.354,A -85,B 0,C 180,E1 -7118.514,E2 -7118.514} C_VEL
LIN {X 0,Y 474.696,Z 144.353,A -85,B 0,C 180,E1 -7121.962,E2 -7121.962} C_VEL
LIN {X 0,Y 474.69,Z 144.359,A -85,B 0,C 180,E1 -7125.455,E2 -7125.455} C_VEL
LIN {X 0,Y 474.605,Z 144.365,A -85,B 0,C 180,E1 -7129.012,E2 -7129.012} C_VEL
LIN {X 0,Y 474.576,Z 144.368,A -85,B 0,C 180,E1 -7131.729,E2 -7131.729} C_VEL
LIN {X 0,Y 474.625,Z 144.359,A -85,B 0,C 180,E1 -7134.494,E2 -7134.494} C_VEL
LIN {X 0,Y 474.598,Z 144.37,A -85,B 0,C 180,E1 -7137.325,E2 -7137.325} C_VEL
LIN {X 0,Y 474.58,Z 144.365,A -85,B 0,C 180,E1 -7140.231,E2 -7140.231} C_VEL
LIN {X 0,Y 474.613,Z 144.367,A -85,B 0,C 180,E1 -7143.221,E2 -7143.221} C_VEL
LIN {X 0,Y 474.58,Z 144.365,A -85,B 0,C 180,E1 -7146.323,E2 -7146.323} C_VEL
LIN {X 0,Y 474.619,Z 144.361,A -85,B 0,C 180,E1 -7149.547,E2 -7149.547} C_VEL
LIN {X 0,Y 474.573,Z 144.366,A -85,B 0,C 180,E1 -7152.229,E2 -7152.229} C_VEL
LIN {X 0,Y 474.613,Z 144.363,A -85,B 0,C 180,E1 -7155.297,E2 -7155.297} C_VEL
LIN {X 0,Y 474.587,Z 144.365,A -85,B 0,C 180,E1 -7158.21,E2 -7158.21} C_VEL
LIN {X 0,Y 474.614,Z 144.364,A -85,B 0,C 180,E1 -7160.451,E2 -7160.451} C_VEL
LIN {X 0,Y 474.577,Z 144.365,A -85,B 0,C 180,E1 -7163.675,E2 -7163.675} C_VEL
LIN {X 0,Y 474.609,Z 144.367,A -85,B 0,C 180,E1 -7166.777,E2 -7166.777} C_VEL
LIN {X 0,Y 474.579,Z 144.365,A -85,B 0,C 180,E1 -7169.768,E2 -7169.768} C_VEL
LIN {X 0,Y 474.596,Z 144.368,A -85,B 0,C 180,E1 -7172.684,E2 -7172.684} C_VEL
LIN {X 0,Y 474.618,Z 144.36,A -85,B 0,C 180,E1 -7175.505,E2 -7175.505} C_VEL
LIN {X 0,Y 474.616,Z 144.362,A -85,B 0,C 180,E1 -7178.887,E2 -7178.887} C_VEL
LIN {X 0,Y 474.623,Z 144.362,A -85,B 0,C 180,E1 -7181.883,E2 -7181.883} C_VEL
LIN {X 0,Y 474.68,Z 144.357,A -85,B 0,C 180,E1 -7184.543,E2 -7184.543} C_VEL
LIN {X 0,Y 474.685,Z 144.358,A -85,B 0,C 180,E1 -7188.037,E2 -7188.037} C_VEL
LIN {X 0,Y 474.657,Z 144.356,A -85,B 0,C 180,E1 -7191.485,E2 -7191.485} C_VEL
LIN {X 0,Y 474.731,Z 144.354,A -85,B 0,C 180,E1 -7194.052,E2 -7194.052} C_VEL
LIN {X 0,Y 474.864,Z 144.331,A -85,B 0,C 180,E1 -7197.455,E2 -7197.455} C_VEL
LIN {X 0,Y 474.871,Z 144.336,A -85,B 0,C 180,E1 -7200,E2 -7200} C_VEL
LIN {X 0,Y 474.863,Z 144.33,A -85,B 0,C 180,E1 -7202.545,E2 -7202.545} C_VEL
LIN {X 0,Y 474.727,Z 144.353,A -85,B 0,C 180,E1 -7205.948,E2 -7205.948} C_VEL
LIN {X 0,Y 474.656,Z 144.356,A -85,B 0,C 180,E1 -7208.515,E2 -7208.515} C_VEL
LIN {X 0,Y 474.684,Z 144.356,A -85,B 0,C 180,E1 -7211.963,E2 -7211.963} C_VEL
LIN {X 0,Y 474.679,Z 144.358,A -85,B 0,C 180,E1 -7215.456,E2 -7215.456} C_VEL
LIN {X 0,Y 474.595,Z 144.365,A -85,B 0,C 180,E1 -7219.013,E2 -7219.013} C_VEL
LIN {X 0,Y 474.567,Z 144.371,A -85,B 0,C 180,E1 -7221.73,E2 -7221.73} C_VEL
LIN {X 0,Y 474.614,Z 144.36,A -85,B 0,C 180,E1 -7224.495,E2 -7224.495} C_VEL
LIN {X 0,Y 474.589,Z 144.371,A -85,B 0,C 180,E1 -7227.327,E2 -7227.327} C_VEL
LIN {X 0,Y 474.542,Z 144.369,A -85,B 0,C 180,E1 -7230.235,E2 -7230.235} C_VEL
LIN {X 0,Y 474.606,Z 144.369,A -85,B 0,C 180,E1 -7233.223,E2 -7233.223} C_VEL
LIN {X 0,Y 474.565,Z 144.367,A -85,B 0,C 180,E1 -7236.326,E2 -7236.326} C_VEL
LIN {X 0,Y 474.593,Z 144.365,A -85,B 0,C 180,E1 -7239.644,E2 -7239.644} C_VEL
LIN {X 0,Y 474.569,Z 144.366,A -85,B 0,C 180,E1 -7242.231,E2 -7242.231} C_VEL
LIN {X 0,Y 474.607,Z 144.365,A -85,B 0,C 180,E1 -7245.299,E2 -7245.299} C_VEL
LIN {X 0,Y 474.585,Z 144.365,A -85,B 0,C 180,E1 -7248.212,E2 -7248.212} C_VEL
LIN {X 0,Y 474.612,Z 144.363,A -85,B 0,C 180,E1 -7250.452,E2 -7250.452} C_VEL
LIN {X 0,Y 474.565,Z 144.367,A -85,B 0,C 180,E1 -7253.675,E2 -7253.675} C_VEL
LIN {X 0,Y 474.608,Z 144.369,A -85,B 0,C 180,E1 -7256.778,E2 -7256.778} C_VEL
LIN {X 0,Y 474.546,Z 144.37,A -85,B 0,C 180,E1 -7259.767,E2 -7259.767} C_VEL
LIN {X 0,Y 474.599,Z 144.369,A -85,B 0,C 180,E1 -7262.685,E2 -7262.685} C_VEL
LIN {X 0,Y 474.621,Z 144.568,A -85,B 0,C 180,E1 -7264.591,E2 -7264.591} C_VEL
LIN {X 0,Y 476.574,Z 154.694,A -85,B 0,C 180,E1 -7266.537,E2 -7266.537} C_VEL
LIN {X 0,Y 476.409,Z 164.715,A -85,B 0,C 180,E1 -7268.339,E2 -7268.339} C_VEL
LIN {X 0,Y 475.668,Z 182.54,A -85,B 0,C 180,E1 -7271.479,E2 -7271.479} C_VEL
LIN {X 0,Y 475.328,Z 192.835,A -85,B 0,C 180,E1 -7273.275,E2 -7273.275} C_VEL
LIN {X 0,Y 477.911,Z 211.158,A -85,B 0,C 180,E1 -7273.67,E2 -7273.67} C_VEL
LIN {X 0,Y 477.148,Z 301.897,A -85,B 0,C 180,E1 -7275.145,E2 -7275.145} C_VEL
LIN {X 0,Y 476.754,Z 315.443,A -85,B 0,C 180,E1 -7275.542,E2 -7275.542} C_VEL
LIN {X 0,Y 476.377,Z 327.757,A -85,B 0,C 180,E1 -7276.075,E2 -7276.075} C_VEL
LIN {X 0,Y 475.886,Z 340.249,A -85,B 0,C 180,E1 -7276.811,E2 -7276.811} C_VEL
LIN {X 0,Y 475.457,Z 351.852,A -85,B 0,C 180,E1 -7277.691,E2 -7277.691} C_VEL
LIN {X 0,Y 475.041,Z 362.36,A -85,B 0,C 180,E1 -7278.696,E2 -7278.696} C_VEL
LIN {X 0,Y 474.576,Z 371.45,A -85,B 0,C 180,E1 -7279.764,E2 -7279.764} C_VEL
LIN {X 0,Y 474.258,Z 380.324,A -85,B 0,C 180,E1 -7281.049,E2 -7281.049} C_VEL
LIN {X 0,Y 474.028,Z 387.401,A -85,B 0,C 180,E1 -7282.333,E2 -7282.333} C_VEL
LIN {X 0,Y 473.866,Z 392.851,A -85,B 0,C 180,E1 -7283.561,E2 -7283.561} C_VEL
LIN {X 0,Y 473.824,Z 397.492,A -85,B 0,C 180,E1 -7284.895,E2 -7284.895} C_VEL
LIN {X 0,Y 473.732,Z 399.831,A -85,B 0,C 180,E1 -7285.747,E2 -7285.747} C_VEL
LIN {X 0,Y 473.794,Z 401.738,A -85,B 0,C 180,E1 -7286.599,E2 -7286.599} C_VEL
LIN {X 0,Y 473.741,Z 403.169,A -85,B 0,C 180,E1 -7287.45,E2 -7287.45} C_VEL
LIN {X 0,Y 473.689,Z 404.799,A -85,B 0,C 180,E1 -7289.151,E2 -7289.151} C_VEL
LIN {X 0,Y 473.672,Z 405.018,A -85,B 0,C 180,E1 -7290.001,E2 -7290.001} C_VEL
LIN {X 0,Y 473.69,Z 404.795,A -85,B 0,C 180,E1 -7290.851,E2 -7290.851} C_VEL
LIN {X 0,Y 473.741,Z 403.146,A -85,B 0,C 180,E1 -7292.552,E2 -7292.552} C_VEL
LIN {X 0,Y 473.795,Z 401.712,A -85,B 0,C 180,E1 -7293.402,E2 -7293.402} C_VEL
LIN {X 0,Y 473.76,Z 398.705,A -85,B 0,C 180,E1 -7294.681,E2 -7294.681} C_VEL
LIN {X 0,Y 473.824,Z 394.638,A -85,B 0,C 180,E1 -7295.96,E2 -7295.96} C_VEL
LIN {X 0,Y 474.013,Z 388.377,A -85,B 0,C 180,E1 -7297.455,E2 -7297.455} C_VEL
LIN {X 0,Y 474.245,Z 381.548,A -85,B 0,C 180,E1 -7298.738,E2 -7298.738} C_VEL
LIN {X 0,Y 474.513,Z 373.066,A -85,B 0,C 180,E1 -7300.023,E2 -7300.023} C_VEL
LIN {X 0,Y 474.97,Z 364.328,A -85,B 0,C 180,E1 -7301.091,E2 -7301.091} C_VEL
LIN {X 0,Y 475.391,Z 354.015,A -85,B 0,C 180,E1 -7302.121,E2 -7302.121} C_VEL
LIN {X 0,Y 475.781,Z 342.904,A -85,B 0,C 180,E1 -7303.019,E2 -7303.019} C_VEL
LIN {X 0,Y 476.285,Z 331.035,A -85,B 0,C 180,E1 -7303.766,E2 -7303.766} C_VEL
LIN {X 0,Y 476.724,Z 318.747,A -85,B 0,C 180,E1 -7304.351,E2 -7304.351} C_VEL
LIN {X 0,Y 477.053,Z 306.281,A -85,B 0,C 180,E1 -7304.777,E2 -7304.777} C_VEL
LIN {X 0,Y 477.36,Z 292.131,A -85,B 0,C 180,E1 -7305.068,E2 -7305.068} C_VEL
LIN {X 0,Y 478.002,Z 209.295,A -85,B 0,C 180,E1 -7306.418,E2 -7306.418} C_VEL
LIN {X 0,Y 475.27,Z 192.073,A -85,B 0,C 180,E1 -7306.816,E2 -7306.816} C_VEL
LIN {X 0,Y 475.804,Z 175.797,A -85,B 0,C 180,E1 -7309.614,E2 -7309.614} C_VEL
LIN {X 0,Y 476.338,Z 161.461,A -85,B 0,C 180,E1 -7312.101,E2 -7312.101} C_VEL
LIN {X 0,Y 476.528,Z 155.004,A -85,B 0,C 180,E1 -7313.237,E2 -7313.237} C_VEL
LIN {X 0,Y 474.623,Z 144.368,A -85,B 0,C 180,E1 -7315.249,E2 -7315.249} C_VEL
LIN {X 0,Y 474.591,Z 144.368,A -85,B 0,C 180,E1 -7318.287,E2 -7318.287} C_VEL
LIN {X 0,Y 474.577,Z 144.372,A -85,B 0,C 180,E1 -7321.22,E2 -7321.22} C_VEL
LIN {X 0,Y 474.62,Z 144.362,A -85,B 0,C 180,E1 -7324.243,E2 -7324.243} C_VEL
LIN {X 0,Y 474.544,Z 144.374,A -85,B 0,C 180,E1 -7327.389,E2 -7327.389} C_VEL
LIN {X 0,Y 474.603,Z 144.364,A -85,B 0,C 180,E1 -7329.644,E2 -7329.644} C_VEL
LIN {X 0,Y 474.572,Z 144.372,A -85,B 0,C 180,E1 -7332.94,E2 -7332.94} C_VEL
LIN {X 0,Y 474.604,Z 144.36,A -85,B 0,C 180,E1 -7335.894,E2 -7335.894} C_VEL
LIN {X 0,Y 474.593,Z 144.363,A -85,B 0,C 180,E1 -7339.34,E2 -7339.34} C_VEL
LIN {X 0,Y 474.597,Z 144.361,A -85,B 0,C 180,E1 -7341.707,E2 -7341.707} C_VEL
LIN {X 0,Y 474.62,Z 144.367,A -85,B 0,C 180,E1 -7344.725,E2 -7344.725} C_VEL
LIN {X 0,Y 474.629,Z 144.361,A -85,B 0,C 180,E1 -7347.787,E2 -7347.787} C_VEL
LIN {X 0,Y 474.596,Z 144.365,A -85,B 0,C 180,E1 -7350.892,E2 -7350.892} C_VEL
LIN {X 0,Y 474.592,Z 144.364,A -85,B 0,C 180,E1 -7353.624,E2 -7353.624} C_VEL
LIN {X 0,Y 474.638,Z 144.36,A -85,B 0,C 180,E1 -7356.642,E2 -7356.642} C_VEL
LIN {X 0,Y 474.651,Z 144.361,A -85,B 0,C 180,E1 -7360.09,E2 -7360.09} C_VEL
LIN {X 0,Y 474.596,Z 144.365,A -85,B 0,C 180,E1 -7362.773,E2 -7362.773} C_VEL
LIN {X 0,Y 474.64,Z 144.361,A -85,B 0,C 180,E1 -7365.421,E2 -7365.421} C_VEL
LIN {X 0,Y 474.708,Z 144.356,A -85,B 0,C 180,E1 -7368.038,E2 -7368.038} C_VEL
LIN {X 0,Y 474.7,Z 144.356,A -85,B 0,C 180,E1 -7371.486,E2 -7371.486} C_VEL
LIN {X 0,Y 474.742,Z 144.352,A -85,B 0,C 180,E1 -7374.052,E2 -7374.052} C_VEL
LIN {X 0,Y 474.877,Z 144.335,A -85,B 0,C 180,E1 -7377.455,E2 -7377.455} C_VEL
LIN {X 0,Y 474.887,Z 144.335,A -85,B 0,C 180,E1 -7380,E2 -7380} C_VEL
LIN {X 0,Y 474.888,Z 144.332,A -85,B 0,C 180,E1 -7382.545,E2 -7382.545} C_VEL
LIN {X 0,Y 474.739,Z 144.352,A -85,B 0,C 180,E1 -7386.375,E2 -7386.375} C_VEL
LIN {X 0,Y 474.71,Z 144.357,A -85,B 0,C 180,E1 -7386.642,E2 -7386.642} C_VEL
LIN {X 0,Y 475.807,Z 150.568,A -85,B 0,C 180,E1 -7387.877,E2 -7387.877} C_VEL
LIN {X 0,Y 475.705,Z 160.628,A -85,B 0,C 180,E1 -7389.782,E2 -7389.782} C_VEL
LIN {X 0,Y 475.524,Z 168.369,A -85,B 0,C 180,E1 -7391.239,E2 -7391.239} C_VEL
LIN {X 0,Y 478.251,Z 182.946,A -85,B 0,C 180,E1 -7391.604,E2 -7391.604} C_VEL
LIN {X 0,Y 477.27,Z 276.698,A -85,B 0,C 180,E1 -7393.155,E2 -7393.155} C_VEL
LIN {X 0,Y 476.967,Z 290.321,A -85,B 0,C 180,E1 -7393.561,E2 -7393.561} C_VEL
LIN {X 0,Y 476.634,Z 303.243,A -85,B 0,C 180,E1 -7394.136,E2 -7394.136} C_VEL
LIN {X 0,Y 476.212,Z 315.271,A -85,B 0,C 180,E1 -7394.858,E2 -7394.858} C_VEL
LIN {X 0,Y 475.768,Z 326.187,A -85,B 0,C 180,E1 -7395.693,E2 -7395.693} C_VEL
LIN {X 0,Y 475.315,Z 336.211,A -85,B 0,C 180,E1 -7396.648,E2 -7396.648} C_VEL
LIN {X 0,Y 474.969,Z 344.868,A -85,B 0,C 180,E1 -7397.658,E2 -7397.658} C_VEL
LIN {X 0,Y 474.599,Z 352.576,A -85,B 0,C 180,E1 -7398.744,E2 -7398.744} C_VEL
LIN {X 0,Y 474.251,Z 360.676,A -85,B 0,C 180,E1 -7400.154,E2 -7400.154} C_VEL
LIN {X 0,Y 474.071,Z 365.944,A -85,B 0,C 180,E1 -7401.306,E2 -7401.306} C_VEL
LIN {X 0,Y 473.903,Z 370.941,A -85,B 0,C 180,E1 -7402.68,E2 -7402.68} C_VEL
LIN {X 0,Y 473.786,Z 374.692,A -85,B 0,C 180,E1 -7404.075,E2 -7404.075} C_VEL
LIN {X 0,Y 473.633,Z 377.271,A -85,B 0,C 180,E1 -7405.488,E2 -7405.488} C_VEL
LIN {X 0,Y 473.619,Z 378.801,A -85,B 0,C 180,E1 -7407.083,E2 -7407.083} C_VEL
LIN {X 0,Y 473.629,Z 378.824,A -85,B 0,C 180,E1 -7408.897,E2 -7408.897} C_VEL
LIN {X 0,Y 473.72,Z 377.126,A -85,B 0,C 180,E1 -7410.629,E2 -7410.629} C_VEL
LIN {X 0,Y 473.809,Z 373.889,A -85,B 0,C 180,E1 -7412.276,E2 -7412.276} C_VEL
LIN {X 0,Y 473.922,Z 369.213,A -85,B 0,C 180,E1 -7413.854,E2 -7413.854} C_VEL
LIN {X 0,Y 474.108,Z 363.312,A -85,B 0,C 180,E1 -7415.319,E2 -7415.319} C_VEL
LIN {X 0,Y 474.377,Z 356.596,A -85,B 0,C 180,E1 -7416.618,E2 -7416.618} C_VEL
LIN {X 0,Y 474.73,Z 348.301,A -85,B 0,C 180,E1 -7417.907,E2 -7417.907} C_VEL
LIN {X 0,Y 475.128,Z 338.847,A -85,B 0,C 180,E1 -7419.088,E2 -7419.088} C_VEL
LIN {X 0,Y 475.532,Z 328.672,A -85,B 0,C 180,E1 -7420.111,E2 -7420.111} C_VEL
LIN {X 0,Y 475.954,Z 317.861,A -85,B 0,C 180,E1 -7420.99,E2 -7420.99} C_VEL
LIN {X 0,Y 476.449,Z 306.24,A -85,B 0,C 180,E1 -7421.731,E2 -7421.731} C_VEL
LIN {X 0,Y 476.757,Z 293.712,A -85,B 0,C 180,E1 -7422.338,E2 -7422.338} C_VEL
LIN {X 0,Y 477.072,Z 280.558,A -85,B 0,C 180,E1 -7422.787,E2 -7422.787} C_VEL
LIN {X 0,Y 477.302,Z 265.533,A -85,B 0,C 180,E1 -7423.085,E2 -7423.085} C_VEL
LIN {X 0,Y 477.467,Z 243.374,A -85,B 0,C 180,E1 -7423.435,E2 -7423.435} C_VEL
LIN {X 0,Y 476.849,Z 237.574,A -85,B 0,C 180,E1 -7423.548,E2 -7423.548} C_VEL
LIN {X 0,Y 471.527,Z 218.891,A -85,B 0,C 180,E1 -7424.025,E2 -7424.025} C_VEL
LIN {X 0,Y 470.929,Z 213.093,A -85,B 0,C 180,E1 -7424.14,E2 -7424.14} C_VEL
LIN {X 0,Y 471.153,Z 183.023,A -85,B 0,C 180,E1 -7424.639,E2 -7424.639} C_VEL
